(* CoDeSys 2.3.9.50 project: flat.pro *)
(* Libraries: COMlibV2.lb6 25.2.14 08:37:08, TcpIp.lib 9.1.14 13:33:22, TcBase.lib 14.5.09 11:14:08, TcSystem.lib 7.6.16 10:01:22, ModbusRTU.lib 13.5.15 12:38:16, TcIoFunctions.lib 27.1.17 16:22:22, TcUtilities.lib 3.2.16 15:08:58, STANDARD.LIB 5.6.98 11:03:02 *)

(* Task configuration *)
TASK Standard (PRIORITY := 0, INTERVAL := T#50ms);
	MAIN
END_TASK

(* Global variable list: Global_Variables *)
VAR_GLOBAL

	Clear						: ClearComBuffer;
	MB							: ModbusRtuMaster_KL6x22B;
	TxBufferCom1				: ComBuffer;
	RxBufferCom1				: ComBuffer;
	SerialLineControlCom1			: SerialLineControl;
	ReceiveDataCom1			: ReceiveData;
	SendDataCom1				: SendData;

	iobroker	: iobroker_Struct;
	mqtt_set:			ST_MqttSettings;


	HW_trans_power						AT	%QX0.1:BOOL:=FALSE; (*Подача тока на трансформатор и реле ТЭН-а *)
	HW_vent_in_heat						AT	%QX0.2:BOOL:=FALSE; (* Подогрев притока - ТЭН *)

	HW_vent_in_trans_105_130				AT	%QX0.3:BOOL:=FALSE;  (* Напряжение 110 или 130 В *)
	HW_vent_in_trans_160_220				AT	%QX0.4:BOOL:=TRUE;  (* Напряжение 160 или 220 В *)
	HW_vent_in_trans_LO_HI				AT	%QX0.5:BOOL:=FALSE;  (* Напряжение 110/130  или 160/220 В *)
	HW_steam							AT	%QX0.6:BOOL:=FALSE; (* Разрешение включения увлажнителя *)

	HW_vent_out							AT	%QX0.7:BOOL:=FALSE; (* Вытяжной вентилятор*)
	HW_kitchen_vent_out					AT	%QX1.0:BOOL:=FALSE; (*Надплитная вытяжка*)
	HW_vent_in_heat_level				AT	%QX1.1:BOOL:=FALSE; (* Подогрев притока ночной режим   -5 К ТЭН *)
	HW_vent_valve						AT	%QX1.2:BOOL:=FALSE; (*Клапан приточной вентиляции"*)

	HW_valve_water_kitchen				AT	%QX1.3:BOOL; (* Кран ХВС и ГВС на кухне *)
	HW_valve_water_bathroom				AT	%QX1.4:BOOL; (* Кран ХВС и ГВС в санузле *)
	HW_LIGHT_ALL						AT	%QX1.5:BOOL; (*Свет в квартире *)
	HW_LIGHT_hall						AT	%QX1.6:BOOL:=FALSE; (*Ночной/аварийный свет в коридоре *)


	HW_sensor_fld_kitchen				AT %IX0.0:BOOL; (* Датчик протечки на кухне*)
	HW_sensor_fld_tlt						AT %IX0.1:BOOL; (* Датчик протечки в туалете*)
	HW_sensor_fld_post					AT %IX0.2:BOOL; (* Датчик протечки в постирочной*)
	HW_sensor_fld_van					AT %IX0.3:BOOL; (* Датчик протечки в ванной*)
	HW_impulse_kitchen_water_warm		AT %IX0.5:BOOL; (* Счётчик горячей воды на кухне*)
	HW_impulse_kitchen_water_cold		AT %IX0.4:BOOL; (* Счётчик холодной воды на кухне*)
	HW_vent_reay_pressure				AT %IX0.6:BOOL; (*Реле давления*)
	HW_kitchen_button_vent_out			AT %IX0.7:BOOL; (* Кнопка кухонной вытяжки*)

	HW_sensor_vent_valve_opened		AT %IX1.0:BOOL;
	HW_sensor_vent_valve_closed			AT %IX1.1:BOOL;
	HW_impulse_bathroom_water_cold		AT %IX1.2:BOOL; (* Счётчик горячей воды санузла NAMUR*)
	HW_impulse_bathroom_water_warm		AT %IX1.3:BOOL; (* Счётчик холодной воды санузла NAMUR*)
	HW_IN01							AT %IX1.4:BOOL;(*Кнопка вкл и откл света в квартире*)
	HW_IN02							AT %IX1.5:BOOL;(*Кнопка вкл и откл кранов воды на кухне*)
	HW_IN03							AT %IX1.6:BOOL;(*Кнопка вкл и откл кранов воды на кухне*)
	HW_IN04							AT %IX1.7:BOOL;(*Кнопка вкл и откл Вентиляции*)
	HW_IN05							AT %IX2.0:BOOL;(*Кнопка вкл и откл Резерв*)

	HW_gerkon							AT %IX2.1:BOOL;(*Датчик открытия двери - геркон*)
	HW_PIR_door						AT %IX2.2:BOOL;(*Датчик открытия двери - pir *)
	HW_PIR_hall							AT %IX2.3:BOOL;(*Датчик открытия двери - pir *)



	HW_vent_out_level					AT	%QW4:WORD:=7000;(* Напряжение управления вытяжным вентилятором (0-32767) *)

	HW_temp_kitchen_box					AT %IW32:WORD; (*Температура на кухне в коробе  *)
	HW_temp_vent_in						AT %IW34:WORD; (*Температура притока перед фильтром *)
	HW_temp_street						AT %IW36:WORD; (*Температура на улице *)
	HW_temp_bedroom					AT %IW38:WORD; (*Температура в спальне *)


END_VAR

(* Global variable list: Global_Variables_persistent *)
VAR_GLOBAL PERSISTENT

	(*USER VARIABLES NEED TO BE ATTACHED TO %Q TO ENABLE SAVE IT IN NOVRAM, FOR CX ONLY *)

	Target_hum_mem		AT %Q*:		INT;
	Target_CO2_mem		AT %Q*:		INT;
	Vent_mem			AT %Q*:		BOOL;
	Vent_out_mem		AT %Q*:		BOOL;
	Vent_heat_mem		AT %Q*:		INT;
	Steam_mem			AT %Q*:		BOOL;
	Vent_heat_level_mem	AT %Q*:		BOOL;
	Light_mem			AT %Q*:		BOOL; (*Свет в квартире*)

	Kitchen_stat_cold_water_mem		AT %Q*:		DINT;
	Kitchen_stat_warm_water_mem		AT %Q*:		DINT;
	Bathroom_stat_cold_water_mem		AT %Q*:		DINT;
	Bathroom_stat_warm_water_mem	AT %Q*:		DINT;


END_VAR

(* Global variable list: TwinCAT_Configuration *)
(* Generated automatically by TwinCAT - (read only) *)
VAR_CONFIG
	.Target_hum_mem AT %QB36 : INT;
	.Target_CO2_mem AT %QB38 : INT;
	.Vent_mem AT %QX60.0 : BOOL;
	.Vent_out_mem AT %QX60.1 : BOOL;
	.Vent_heat_mem AT %QB40 : INT;
	.Steam_mem AT %QX60.2 : BOOL;
	.Vent_heat_level_mem AT %QX60.3 : BOOL;
	.Light_mem AT %QX60.4 : BOOL;
	.Kitchen_stat_cold_water_mem AT %QB44 : DINT;
	.Kitchen_stat_warm_water_mem AT %QB48 : DINT;
	.Bathroom_stat_cold_water_mem AT %QB52 : DINT;
	.Bathroom_stat_warm_water_mem AT %QB56 : DINT;
END_VAR

(* Global variable list: Variable_Configuration *)
VAR_CONFIG
	MB.InData AT %IB12 : MB_KL6inData22B;
	MB.OutData AT %QB12 : MB_KL6outData22B;
END_VAR

(* Data type *)
TYPE iobroker_Struct  :
STRUCT
	Vent_status				: 	INT;
	Valve_status				: 	INT;
	Kitchen_room_temp 		:	REAL;
	Kitchen_room_hum 		:	REAL;
	Kitchen_room_CO2		:	REAL;

	Child_small_room_temp 	:	REAL;
	Child_small_room_hum 	:	REAL;
	Child_small_room_CO2 	:	REAL;

	Child_big_room_temp	 	:	REAL;
	Child_big_room_hum	 	:	REAL;
	Child_big_room_CO2	 	:	REAL;

	Bed_room_temp	 		:	REAL;
	Bed_room_temp2	 		:	REAL;
	Bed_room_hum	 		:	REAL;
	Bed_room_hum2	 		:	REAL;
	Bed_room_CO2			:	REAL;

	Kitchen_room_tempout		:	REAL;
	Kitchen_room_tempout_2	:	REAL;

	FLD_valve_kitchen 		:	BOOL; (* Положение  крана воды на кухне*)
	FLD_valve_bathroom 		:	BOOL; (*Положение  крана воды в санузле*)
	FLD_PRC				:	BOOL; (*Датчик в постирочной*)
	FLD_TLT				:	BOOL; (*Датчик в туалете*)
	FLD_BATH				:	BOOL;(*Датчик в  ванной*)
	FLD_KUH				:	BOOL;(*Датчик на  кухне*)
	FLD_ALRM_KITCHEN 		:	BOOL; (*ТРЕВОГА ЗАТОПЛЕНИЕ НА КУХНЕ*)
	FLD_ALRM_BATH 		:	BOOL; (*ТРЕВОГА ЗАТОПЛЕНИЕ В САНУЗЛЕ*)


	Kitchen_stat_cold_water	:	DINT;
	Kitchen_stat_warm_water	:	DINT;
	Bathroom_stat_cold_water	:	DINT;
	Bathroom_stat_warm_water	:	DINT;

	Steam_status				:	INT;
	Steam_real				:	INT;

	Vent_input_level			:	INT;  (*  0-220 V  *)
	Vent_output_level			:	INT; (*0-100%*)
	Soft_kitchen_button_vent_out:	BOOL; (*Вирутальная  кнопка кухонной вытяжки*)

	Temp_vent_in			:	REAL;
	Vent_pressure_relay		:	BOOL;

	PT_temp_bedroom		:	REAL;
	Vent_valve_status			:	INT;


	(* SETTINGS *)
	Rezerv					:	BOOL;
	Steam_level				:	INT;
	Security_status			:	INT;
	Target_hum				:	INT;
	Target_CO2				:	INT;
	Vent						:	BOOL;
	Vent_out					:	BOOL;
	Vent_heat				:	INT;
	Steam					:	BOOL;
	Vent_heat_level			:	BOOL;
	Light					:	BOOL; (*Свет в квартире*)
	Light_hall				:	BOOL; (*Свет в коридоре*)
	Gerkon					:	BOOL; (*Датчик открытия входной двери (геркон)*)
	PIR_door				:	BOOL;(*Датчик открытия входной двери PIR-штора*)

	Uv						:	REAL;
	Ia						:	REAL;
	Pw						:	REAL;
	E_T1					:	REAL;
	E_T2					:	REAL;
	E_T4					:	REAL;

END_STRUCT
END_TYPE

(* Data type *)
(* @NESTEDCOMMENTS := 'Yes' *)
(* @PATH := '' *)
(* @OBJECTFLAGS := '0, 8' *)
TYPE ST_MqttReceivedPublishTelegram :
STRUCT
	sTopic		: STRING[255];
	sValue		: STRING[255];
	bHasData	: BOOL;
END_STRUCT
END_TYPE
(* @END_DECLARATION := '0' *)

(* Data type *)
(* @NESTEDCOMMENTS := 'Yes' *)
(* @PATH := '' *)
(* @OBJECTFLAGS := '0, 8' *)
TYPE ST_MqttSettings :
STRUCT
	(* informations *)
(*	sMqttClientId	: STRING[23]:='plc';
	sMqttUserId	: STRING[25]:='mqtt';
	sMqttPassword	: STRING[25]:='mqtt';
	sMqttBrokerIP	: STRING[15]:='192.168.3.200';
	nMqttBrokerPort	: UDINT := 1883;

	(* state *)
	bSocketConnection	: BOOL := FALSE;
	bConnected			: BOOL := FALSE;
	bConnectPackageSent	: BOOL := FALSE;
	bDisconnect			: BOOL := FALSE;
	bError				: BOOL := FALSE;
	bValidConnection	: BOOL := FALSE;
	bActive				: BOOL := FALSE;
	wPackageIdentifier	: WORD := 1;
	hSocket				: T_HSOCKET;
	tonSendPingReq		: TON;

	(* send *)
	stMqttSendTelegram			: ST_MqttTelegram;
	stMqttLastSendTelegram		: ST_MqttTelegram;

	(* receive *)
	stMqttReceivedTelegram			: ST_MqttTelegram;
	stMqttLastReceivedTelegram		: ST_MqttTelegram;
	stMqttReceivedPublishTelegram	: ST_MqttReceivedPublishTelegram;

	(* settings internal *)
	iTelegramSize	: INT := 544;
	usKeepAliveTime	: USINT := 60; (* seconds *)

*)



	(* informations *)
	sMqttClientId	: STRING[23];
	sMqttUserId	: STRING[25];
	sMqttPassword	: STRING[25];
	sMqttBrokerIP	: STRING[15];
	nMqttBrokerPort	: UDINT := 1883;

	(* state *)
	bSocketConnection	: BOOL := FALSE;
	bConnected			: BOOL := FALSE;
	bConnectPackageSent	: BOOL := FALSE;
	bDisconnect			: BOOL := FALSE;
	bError				: BOOL := FALSE;
	bValidConnection	: BOOL := FALSE;
	bActive				: BOOL := FALSE;
	wPackageIdentifier	: WORD := 1;
	hSocket				: T_HSOCKET;
	tonSendPingReq		: TON;

	(* send *)
	stMqttSendTelegram			: ST_MqttTelegram;
	stMqttLastSendTelegram		: ST_MqttTelegram;

	(* receive *)
	stMqttReceivedTelegram			: ST_MqttTelegram;
	stMqttLastReceivedTelegram		: ST_MqttTelegram;
	stMqttReceivedPublishTelegram	: ST_MqttReceivedPublishTelegram;

	(* settings internal *)
	iTelegramSize	: INT := 544;
	usKeepAliveTime	: USINT := 60; (* seconds *)










END_STRUCT
END_TYPE
(* @END_DECLARATION := '0' *)

(* Data type *)
(* @NESTEDCOMMENTS := 'Yes' *)
(* @PATH := '' *)
(* @OBJECTFLAGS := '0, 8' *)
TYPE ST_MqttTelegram :
STRUCT
	arMqttData 	: ARRAY[0..544] OF BYTE;
	nDataLength	: UDINT := 0;
END_STRUCT
END_TYPE
(* @END_DECLARATION := '0' *

(* POU MAIN, ST *)
PROGRAM MAIN
VAR
	INITVAR					: BOOL:=FALSE;
	SW_LIGHT				: SM_BUTT;		(* вкл/откл  света в квартире *)
	SW_VENT				: SM_BUTT;		(* вкл/откл вентиляции *)
	SW_REZERV			: SM_BUTT;





END_VAR
IF (INITVAR=FALSE) THEN

(* RESTORE VARS FROM MEMORY AFTER REBOOT/RESET/LOST POWER *)

	iobroker.Target_hum		:=	Target_hum_mem;
	iobroker.Target_CO2		:=	Target_CO2_mem;
	iobroker.Vent				:=	Vent_mem;
	iobroker.Vent_out			:=	Vent_out_mem;
	iobroker.Vent_heat		:=	Vent_heat_mem;
	iobroker.Steam			:=	Steam_mem;
	iobroker.Vent_heat_level	:=	Vent_heat_level_mem;
	iobroker.Light				:=	Light_mem;

	iobroker.Kitchen_stat_cold_water		:=	Kitchen_stat_cold_water_mem;
	iobroker.Kitchen_stat_warm_water		:=	Kitchen_stat_warm_water_mem;
	iobroker.Bathroom_stat_cold_water		:=	Bathroom_stat_cold_water_mem;
	iobroker.Bathroom_stat_warm_water		:=	Bathroom_stat_warm_water_mem;

	INITVAR:=TRUE;
ELSE

	(* SAVE VARS to PERSISTENT *)

	Target_hum_mem		:=	iobroker.Target_hum;
	Target_CO2_mem		:=	iobroker.Target_CO2;
	Vent_mem			:=	iobroker.Vent;
	Vent_out_mem		:=	iobroker.Vent_out;
	Vent_heat_mem		:=	iobroker.Vent_heat;
	Steam_mem			:=	iobroker.Steam;
	Vent_heat_level_mem	:=	iobroker.Vent_heat_level;
	Light_mem			:=	iobroker.Light;

	Mqtt;					(*Отправка данных mqtt *)
	Sensors;					(* Аналоговые датчики на модуле KL *)
	RS485read;				(* Работа с устройствами на шине RS485 *)
	VentControl;				(* Глобальный контроль вентустановки*)
	VentPower;				(* Авторегулировка мощности вентустановки по датчикам CO2*)
	Counters;				(* Счётчики воды *)
	Fluid_bath;				(* Защита от протечки в санузлах. Оработка нажатия физической и виртульной кнопки №2 *)
	Fluid_kitchen;				(* Защита от протечки в кухне. Оработка нажатия физической и виртульной кнопки №3 *)
	Light_hall;				(* Свет в коридоре *)



(* Оработка нажатия физических и виртульных кнопок №1, №4, №5 *)

	SW_LIGHT 		(IN:=HW_IN01, IN1:= iobroker.Light, 	Q=>NOT iobroker.Light);	(* Конпка №1 *)
	SW_VENT 		(IN:=HW_IN04, IN1:=iobroker.Vent, 	Q=>iobroker.Vent);		(* Конпка №4 *)
	SW_REZERV 	(IN:=HW_IN05, IN1:=iobroker.Rezerv, 	Q=>iobroker.Rezerv);	(* Конпка №5 *)


(* Прямая связь между экспортирумымми переменными и  переменными, жестко привязаными  к физ. портам. Частота обновления= циклу ПЛК  : *)

	HW_LIGHT_ALL	:=NOT iobroker.Light;					(* СВЕТ в квартире*)
	HW_LIGHT_HALL	:=iobroker.Light_hall;					(* СВЕТ в квартире*)
	iobroker.Gerkon	:=HW_gerkon;						(* Геркон на двери*)
	iobroker.PIR_door:=HW_pir_door;						(* Датчик движения на двери *)
	iobroker.Vent_pressure_relay:=HW_vent_reay_pressure; 	(* Relay pressure *)

END_IF
END_PROGRAM

(* POU SM_BUTT, ST *)
FUNCTION_BLOCK SM_BUTT            (* ФУНКЦИОНАЛЬНЫЙ БЛОК ДЛЯ ПРОСТОЙ КНОПКИ *)
    VAR_INPUT
       	IN: BOOL;          	(*ВХОД ЗА КОТОРЫМ МЫ СЛЕДИМ *)
	IN1:BOOL;				(*ВЫХОД ЗА КОТОРЫМ ТОЖЕ СЛЕДИМ*)
    END_VAR

    VAR_OUTPUT
	Q : BOOL;        			(*СОСТОЯНИЕ ВЫХОДА*)
    END_VAR
    VAR
  MEM : BOOL;    			(* ВНУТРЕННЯЯ ПЕРЕМЕННАЯ ДЛЯ ХРАНЕНИЯ СОСТОЯНИЯ КНОПКИ *)
    END_VAR
Q:=IN1;

IF IN AND NOT MEM THEN 	(* ПОЙМАЛИ ПЕРЕДНИЙ ФРОНТ - НАЖАЛИ НА КНОПКУ *)
	Q := NOT IN1;    			(* МЕНЯЕМ СОСТОЯНИЕ ВЫХОДА НА ПРОТИВОПОЛОЖНОЕ *)
END_IF

MEM := IN;                       		(* ЗАПОМИНАЕМ ТЕКУЩЕЕ ЗНАЧЕНИЕ КНОПКИ *)
END_FUNCTION_BLOCK

(* POU Mqtt, ST *)
PROGRAM Mqtt
VAR
	FB_Mqtt_Controller 		: FB_Mqtt_Controller_V10;
	stMqttSettings				: ST_MqttSettings;
	bMqttControllerBusy		: BOOL;
	FB_Mqtt_Publish1 			: FB_Mqtt_Publish_V10;
	FB_Mqtt_Publish2			: FB_Mqtt_Publish_V10;
	FB_Mqtt_Publish3			: FB_Mqtt_Publish_V10;
	FB_Mqtt_Publish4			: FB_Mqtt_Publish_V10;
	bPublishBusy1			: BOOL;
	bPublishBusy2			: BOOL;
	bPublishBusy3			: BOOL;
	bPublishBusy4			: BOOL;
END_VAR
(*        SEND DATA VIA MQTT  *)

FB_Mqtt_Controller (
		bActive			:= TRUE,
		sMqttClientId		:= 'plc',
		sMqttUserId		:= 'mqtt',
		sMqttPassword	:= 'mqtt',
		sMqttBrokerIp		:= '192.168.3.200',
		nMqttBrokerPort	:= 1883,
		stMqttSettings		:= stMqttSettings,
		bBusy			=> bMqttControllerBusy
	);
	IF bMqttControllerBusy THEN
		RETURN;
	END_IF

		FB_Mqtt_Publish1(sTopic:='BECKHOFF_CX9010/CO2/Kitchen',sValue:=REAL_TO_STRING(iobroker.Kitchen_room_CO2),bRetain:=TRUE, stMqttSettings:=stMqttSettings,bBusy => bPublishBusy1 );
		FB_Mqtt_Publish2(sTopic:='BECKHOFF_CX9010/CO2/Bed_room',sValue:=REAL_TO_STRING(iobroker.Bed_room_CO2),bRetain:=TRUE, stMqttSettings:=stMqttSettings,bBusy => bPublishBusy2 );
		FB_Mqtt_Publish3(sTopic:='BECKHOFF_CX9010/CO2/Child_big_room',sValue:=REAL_TO_STRING(iobroker.Child_big_room_CO2),bRetain:=TRUE, stMqttSettings:=stMqttSettings,bBusy => bPublishBusy3 );
		FB_Mqtt_Publish4(sTopic:='BECKHOFF_CX9010/CO2/Child_small_room',sValue:=REAL_TO_STRING(iobroker.Child_small_room_CO2),bRetain:=TRUE, stMqttSettings:=stMqttSettings,bBusy => bPublishBusy4);
END_PROGRAM

(* POU FB_Mqtt_Controller_V10, ST *)
(* @NESTEDCOMMENTS := 'Yes' *)
(* @PATH := '\/_Generic\/Mqtt' *)
(* @OBJECTFLAGS := '0, 8' *)
(* @SYMFILEFLAGS := '2048' *)
FUNCTION_BLOCK FB_Mqtt_Controller_V10
VAR_INPUT
(*	bActive			: BOOL := FALSE;
	sMqttClientId	: STRING[23]:='plc';
	sMqttUserId	: STRING[25] := 'mqtt';
	sMqttPassword	: STRING[25] := 'mqtt';
	sMqttBrokerIP	: STRING[15]:='192.168.3.200';
	nMqttBrokerPort	: UDINT := 1883;
*)
	bActive			: BOOL := FALSE;
	sMqttClientId	: STRING[23];
	sMqttUserId	: STRING[25] := '';
	sMqttPassword	: STRING[25] := '';
	sMqttBrokerIP	: STRING[15];
	nMqttBrokerPort	: UDINT := 1883;
END_VAR
VAR_OUTPUT
	bBusy	: BOOL := FALSE;
END_VAR
VAR_IN_OUT
	stMqttSettings	: ST_MqttSettings;
END_VAR
VAR
	iState			: INT := 0;
	fbSocketConnect	: FB_SocketConnect;
	fbSocketClose	: FB_SocketClose;

	fbMqttTelegramConnect	: FB_MqttTelegram_Connect_V10;
	fbMqttTelegramPingReq	: FB_MqttTelegram_PingReq_V10;
	fbMqttSend				: FB_Mqtt_Send_V10;
	fbMqttReceive			: FB_Mqtt_Receive_V10;
END_VAR
VAR CONSTANT
	C_STARTUP					: INT := 0;
	C_CONNECT					: INT := 100;
	C_CONNECT_WAIT				: INT := 110;
	C_CLOSE						: INT := 200;
	C_CLOSE_WAIT				: INT := 210;
	C_IDLE						: INT := 500;
END_VAR
(* @END_DECLARATION := '0' *)
(*
 * Connects to mqtt broker
 * Sends connect message
 * Sends ping(back)
 * Sends disconnect
 *)
CASE iState OF
	C_STARTUP:
		stMqttSettings.bConnected			:= FALSE;
		stMqttSettings.bConnectPackageSent	:= FALSE;
		stMqttSettings.bDisconnect			:= FALSE;
		stMqttSettings.bSocketConnection	:= FALSE;
		stMqttSettings.bError				:= FALSE;
		stMqttSettings.bValidConnection		:= FALSE;
		stMqttSettings.wPackageIdentifier	:= 1;
		stMqttSettings.bActive				:= bActive;
		stMqttSettings.hSocket				:= fbSocketConnect.hSocket;
		stMqttSettings.nMqttBrokerPort		:= nMqttBrokerPort;
		stMqttSettings.sMqttBrokerIP		:= sMqttBrokerIP;
		stMqttSettings.sMqttClientId		:= sMqttClientId;
		stMqttSettings.sMqttUserId		:= sMqttUserId;
		stMqttSettings.sMqttPassword		:= sMqttPassword;

		stMqttSettings.stMqttReceivedTelegram.nDataLength := 0;

		bBusy := FALSE;

		CallMqttBlocks();

		IF bActive THEN
			iState := C_CONNECT;
		END_IF;

	(* Start connection *)
	C_CONNECT:
		bBusy := TRUE;

		fbSocketConnect(
			bExecute	:= FALSE
		);

		fbSocketConnect(
			sSrvNetId	:= '',
			sRemoteHost	:= sMqttBrokerIP,
			nRemotePort	:= nMqttBrokerPort,
			bExecute	:= TRUE,
			tTimeout	:= USINT_TO_TIME(stMqttSettings.usKeepAliveTime) + t#10s
		);

		iState := C_CONNECT_WAIT;

	(* Wait till connected *)
	C_CONNECT_WAIT:
		fbSocketConnect(
			bExecute := FALSE
		);

		IF
			NOT fbSocketConnect.bBusy
			AND NOT fbSocketConnect.bError
		THEN
			iState 								:= C_IDLE;
			stMqttSettings.hSocket				:= fbSocketConnect.hSocket;
			stMqttSettings.bSocketConnection	:= TRUE;
		END_IF;

		IF fbSocketConnect.bError THEN
			iState := C_STARTUP;
		END_IF;

		IF NOT stMqttSettings.bActive THEN
			iState := C_STARTUP;
		END_IF;

	(* Close connection *)
	C_CLOSE:
		bBusy := TRUE;

		fbSocketClose(
			bExecute	:= TRUE,
			hSocket		:= stMqttSettings.hSocket
		);

		iState := C_CLOSE_WAIT;

	(* Wait close connection *)
	C_CLOSE_WAIT:
		fbSocketClose(
			bExecute := FALSE
		);

		IF
			NOT fbSocketClose.bBusy
			AND NOT fbSocketClose.bError
		THEN
			iState := C_STARTUP;
		END_IF;

		IF fbSocketClose.bError THEN
			iState := C_STARTUP;
		END_IF;

		IF NOT stMqttSettings.bActive THEN
			iState := C_STARTUP;
		END_IF;

	(* Idle *)
	C_IDLE:
		bBusy 					:= FALSE;
		stMqttSettings.bActive	:= bActive;

		stMqttSettings.bValidConnection :=
			NOT stMqttSettings.bError
			AND NOT stMqttSettings.bDisconnect
			AND stMqttSettings.bConnected
			AND stMqttSettings.bSocketConnection
			AND stMqttSettings.bActive;

		CallMqttBlocks();

		IF
			stMqttSettings.bDisconnect
			OR stMqttSettings.bError
			OR NOT stMqttSettings.bActive
		THEN
			IF
				stMqttSettings.bConnected
				OR stMqttSettings.bSocketConnection
			THEN
				(* TODO : send disconnect *)
				iState := C_CLOSE;
			ELSE
				iState := C_CLOSE;
			END_IF;
		END_IF;

	ELSE
		iState := C_STARTUP;
END_CASE;
(*	END_FUNCTION_BLOCK	*)
END_FUNCTION_BLOCK
ACTION CallMqttBlocks:
(*ACTION	CallMqttBlocks: *)
fbMqttReceive(
	stMqttSettings := stMqttSettings
);

fbMqttTelegramConnect(
	stMqttSettings := stMqttSettings
);

fbMqttTelegramPingReq(
	stMqttSettings := stMqttSettings
);

fbMqttSend(
	stMqttSettings := stMqttSettings
);

(* END_ACTION *)
END_ACTION

(* POU Intern/FB_MqttTelegram_Connect_V10, ST *)
(* @NESTEDCOMMENTS := 'Yes' *)
(* @PATH := '\/_Generic\/Mqtt\/Intern' *)
(* @OBJECTFLAGS := '0, 8' *)
(* @SYMFILEFLAGS := '2048' *)
FUNCTION_BLOCK FB_MqttTelegram_Connect_V10
VAR_IN_OUT
	stMqttSettings	: ST_MqttSettings;
END_VAR
VAR
	iState 				: INT := 0;
	idLength			: INT;
	iuLength			: INT;
	ipLength			: INT;
	ipos				: INT;
	stMqttTelegram		: ST_MqttTelegram;
	fbMqttEncodeLength	: FB_Mqtt_EncodeLength_V10;
	bLength1			: BYTE;
	bLength2			: BYTE;
	bLength3			: BYTE;
	bLength4			: BYTE;
	bLengthAmount		: BYTE;
END_VAR
VAR CONSTANT
	C_STARTUP		: INT := 0;
	C_BUILD_CONNECT	: INT := 100;
	C_SEND_WAIT		: INT := 110;
	C_IDLE			: INT := 500;
END_VAR
(* @END_DECLARATION := '0' *)
CASE iState OF
	C_STARTUP:
		IF
			NOT stMqttSettings.bDisconnect
			AND NOT stMqttSettings.bError
			AND stMqttSettings.bSocketConnection
			AND stMqttSettings.bActive
		THEN
			iState := C_IDLE;
		END_IF;

	(* build connect telegram *)
	C_BUILD_CONNECT:
		FC_Mqtt_ClearTelegram_V10(
			stMqttTelegram	:= stMqttTelegram,
			stMqttSettings	:= stMqttSettings
		);

		(* get client id length *)
		idLength := LEN(stMqttSettings.sMqttClientId);
		IF idLength < 1 THEN
			stMqttSettings.sMqttClientId := 'x';
			idLength := 1;
		END_IF;

		IF idLength > 23 THEN
			idLength := 23;
		END_IF;

		IF
			LEN(stMqttSettings.sMqttUserId) > 0
			AND LEN(stMqttSettings.sMqttPassword) > 0
		THEN
			iuLength := LEN(stMqttSettings.sMqttUserId)+2; (* 2 byte data length*)
			ipLength := LEN(stMqttSettings.sMqttPassword)+2; (* 2 byte data length*)
		ELSE
			iuLength := 0;
			ipLength := 0;
		END_IF

		(* Calculate length *)
		(* 10 byte header, 2 byte data length, data length, [user length + 2], [password length + 2]*)
		fbMqttEncodeLength(
			dwLength := 10 + 2 + INT_TO_BYTE(idLength) + INT_TO_BYTE(iuLength) + INT_TO_BYTE(ipLength),
			bLength1 => bLength1,
			bLength2 => bLength2,
			bLength3 => bLength3,
			bLength4 => bLength4,
			bAmount	 => bLengthAmount
		);

		(* MQTT Control Packet type *)
		stMqttTelegram.arMqttData[0] := 16;
		(* Remaining Length *)
		CASE bLengthAmount OF
			1:
				stMqttTelegram.arMqttData[1] := bLength1;

			2:
				stMqttTelegram.arMqttData[1] := bLength1;
				stMqttTelegram.arMqttData[2] := bLength2;

			3:
				stMqttTelegram.arMqttData[1] := bLength1;
				stMqttTelegram.arMqttData[2] := bLength2;
				stMqttTelegram.arMqttData[3] := bLength3;

			4:
				stMqttTelegram.arMqttData[1] := bLength1;
				stMqttTelegram.arMqttData[2] := bLength2;
				stMqttTelegram.arMqttData[3] := bLength3;
				stMqttTelegram.arMqttData[4] := bLength4;
		END_CASE;
		(* init position*)
		ipos := bLengthAmount;

		(* Length MSB *)
		stMqttTelegram.arMqttData[ipos+1] := 0;
		(* Length LSB *)
		stMqttTelegram.arMqttData[ipos+2] := 4;
		(* M *)
		stMqttTelegram.arMqttData[ipos+3] := 77;
		(* Q *)
		stMqttTelegram.arMqttData[ipos+4] := 81;
		(* T *)
		stMqttTelegram.arMqttData[ipos+5] := 84;
		(* T *)
		stMqttTelegram.arMqttData[ipos+6] := 84;
		(* Protocol Level *)
		stMqttTelegram.arMqttData[ipos+7] := 4;
		(* Connect Flags *)
		stMqttTelegram.arMqttData[ipos+8].1 := TRUE;
		stMqttTelegram.arMqttData[ipos+8].6 := (ipLength>2); (* more then 2 byte data length*)
		stMqttTelegram.arMqttData[ipos+8].7 := (iuLength>2); (* more then 2 byte data length*)
		(* Keep Alive MSB *)
		stMqttTelegram.arMqttData[ipos+9] := 0;
		(* Keep Alive LSB *)
		stMqttTelegram.arMqttData[ipos+10] := stMqttSettings.usKeepAliveTime;
		(* Data length MSB *)
		stMqttTelegram.arMqttData[ipos+11] := 0;
		(* Data length LSB *)
		stMqttTelegram.arMqttData[ipos+12] := INT_TO_BYTE(idLength);

		(* Client ID *)
		MEMCPY(
			destAddr	:= ADR(stMqttTelegram.arMqttData[ipos+13]),
		    srcAddr		:= ADR(stMqttSettings.sMqttClientId),
			n  			:= idLength
		);

		ipos := ipos+13+idLength;
		IF (iuLength > 2) THEN (* more then 2 byte data length*)
			(* Data length MSB *)
			stMqttTelegram.arMqttData[ipos] := 0;
			(* Data length LSB *)
			stMqttTelegram.arMqttData[ipos+1] := INT_TO_BYTE(iuLength-2);

			(* User ID *)
			MEMCPY(
				destAddr	:= ADR(stMqttTelegram.arMqttData[ipos+2]),
			    srcAddr		:= ADR(stMqttSettings.sMqttUserId),
				n  			:= iuLength-2
			);
			ipos := ipos+iuLength;
		END_IF

		IF (iuLength > 2) THEN (* more then 2 byte data length*)
			(* Data length MSB *)
			stMqttTelegram.arMqttData[ipos] := 0;
			(* Data length LSB *)
			stMqttTelegram.arMqttData[ipos+1] := INT_TO_BYTE(ipLength-2);

			(* Password *)
			MEMCPY(
				destAddr	:= ADR(stMqttTelegram.arMqttData[ipos+2]),
			    srcAddr		:= ADR(stMqttSettings.sMqttPassword),
				n  			:= ipLength-2
			);
			ipos := ipos+ipLength;
		END_IF

		stMqttTelegram.nDataLength 	:= ipos; (* 1 byte header, 1 byte remaining length *)
		iState 						:= C_SEND_WAIT;

	(* send telegram *)
	C_SEND_WAIT:
		IF stMqttSettings.stMqttSendTelegram.nDataLength = 0 THEN
			FC_Mqtt_CopyTelegram_V10(
				stMqttSrcTelegram	:= stMqttTelegram,
				stMqttDestTelegram	:= stMqttSettings.stMqttSendTelegram,
				stMqttSettings		:= stMqttSettings
			);

			stMqttSettings.bConnectPackageSent	:= TRUE;
			iState								:= C_IDLE;
		END_IF;

		IF
			NOT stMqttSettings.bActive
			OR NOT stMqttSettings.bSocketConnection
		THEN
			iState := C_STARTUP;
		END_IF;

	(* idle *)
	C_IDLE:
		IF
			NOT stMqttSettings.bDisconnect
			AND NOT stMqttSettings.bError
			AND NOT stMqttSettings.bConnected
			AND stMqttSettings.bSocketConnection
			AND NOT stMqttSettings.bConnectPackageSent
			AND stMqttSettings.bActive
		THEN
			iState := C_BUILD_CONNECT;
		END_IF;

		(* check received telegram *)
		IF
			stMqttSettings.bConnectPackageSent
			AND stMqttSettings.stMqttReceivedTelegram.nDataLength = 4
			AND stMqttSettings.stMqttReceivedTelegram.arMqttData[0] = 32
			AND stMqttSettings.stMqttReceivedTelegram.arMqttData[1] = 2
			AND (
				(* Session pressent or not, we ignore *)
				stMqttSettings.stMqttReceivedTelegram.arMqttData[2] = 1
				OR
				stMqttSettings.stMqttReceivedTelegram.arMqttData[2] = 0
			)
			AND stMqttSettings.stMqttReceivedTelegram.arMqttData[3] = 0
		THEN
			stMqttSettings.bConnected := TRUE;
			FC_Mqtt_ClearTelegram_V10(
				stMqttTelegram	:= stMqttSettings.stMqttReceivedTelegram,
				stMqttSettings	:= stMqttSettings
			);
		END_IF;

		(* error on connect *)
		IF
			stMqttSettings.bConnectPackageSent
			AND stMqttSettings.stMqttReceivedTelegram.nDataLength = 4
			AND stMqttSettings.stMqttReceivedTelegram.arMqttData[0] = 32
			AND stMqttSettings.stMqttReceivedTelegram.arMqttData[1] = 2
			AND stMqttSettings.stMqttReceivedTelegram.arMqttData[3] <> 0
		THEN
			stMqttSettings.bError := TRUE;
		END_IF;

		IF
			stMqttSettings.bDisconnect
			OR stMqttSettings.bError
			OR NOT stMqttSettings.bSocketConnection
			OR NOT stMqttSettings.bActive
		THEN
			iState := C_STARTUP;
		END_IF;

	ELSE
		iState := C_STARTUP;
END_CASE;


(*	END_FUNCTION_BLOCK	*)
END_FUNCTION_BLOCK

(* POU Intern/FB_Mqtt_EncodeLength_V10, ST *)
(* @NESTEDCOMMENTS := 'Yes' *)
(* @PATH := '\/_Generic\/Mqtt\/Intern' *)
(* @OBJECTFLAGS := '0, 8' *)
(* @SYMFILEFLAGS := '2048' *)
FUNCTION_BLOCK FB_Mqtt_EncodeLength_V10
VAR_INPUT
	dwLength	: DWORD;
END_VAR
VAR_OUTPUT
	bLength1	: BYTE := 0;
	bLength2	: BYTE := 0;
	bLength3	: BYTE := 0;
	bLength4	: BYTE := 0;
	bAmount		: BYTE := 0;
END_VAR
VAR
	dwWorkLength	: DWORD;
	dwCopyLength	: DWORD;
END_VAR
(* @END_DECLARATION := '0' *)
bAmount 		:= 1;
dwCopyLength	:= dwLength;

WHILE dwCopyLength > 0 DO
	dwWorkLength := dwCopyLength MOD 128;
	dwCopyLength := dwCopyLength / 128;

	IF dwCopyLength > 0 THEN
		dwWorkLength := dwWorkLength OR 128;
	END_IF;

	CASE bAmount OF
		1:
			bLength1 := DWORD_TO_BYTE(dwWorkLength);

		2:
			bLength2 := DWORD_TO_BYTE(dwWorkLength);

		3:
			bLength3 := DWORD_TO_BYTE(dwWorkLength);

		4:
			bLength4 := DWORD_TO_BYTE(dwWorkLength);

		ELSE
			;
	END_CASE;

	IF dwCopyLength > 0 THEN
		bAmount := bAmount + 1;
	END_IF;

	IF bAmount > 4 THEN
		(* hmm *)
		RETURN;
	END_IF;
END_WHILE;
(*
do
	encodedByte = X MOD 128
	X = X DIV 128

	// if there are more data to encode, set the top bit of this byte
	if ( X > 0 )
		encodedByte = encodedByte OR 128
	endif

	'output' encodedByte
while ( X > 0 )
*)

(*	END_FUNCTION_BLOCK	*)
END_FUNCTION_BLOCK

(* POU Intern/FC_Mqtt_ClearTelegram_V10, ST *)
(* @NESTEDCOMMENTS := 'Yes' *)
(* @PATH := '\/_Generic\/Mqtt\/Intern' *)
(* @OBJECTFLAGS := '0, 8' *)
(* @SYMFILEFLAGS := '2048' *)
FUNCTION FC_Mqtt_ClearTelegram_V10 : BOOL
VAR_IN_OUT
	stMqttTelegram	: ST_MqttTelegram;
	stMqttSettings	: ST_MqttSettings;
END_VAR
VAR
END_VAR
(* @END_DECLARATION := '0' *)
MEMSET(
	destAddr	:= ADR(stMqttTelegram.arMqttData),
	fillByte  	:= 0,
	n			:= stMqttSettings.iTelegramSize
);

stMqttTelegram.nDataLength := 0;

(*	END_FUNCTION	*)
END_FUNCTION

(* POU Intern/FC_Mqtt_CopyTelegram_V10, ST *)
(* @NESTEDCOMMENTS := 'Yes' *)
(* @PATH := '\/_Generic\/Mqtt\/Intern' *)
(* @OBJECTFLAGS := '0, 8' *)
(* @SYMFILEFLAGS := '2048' *)
FUNCTION FC_Mqtt_CopyTelegram_V10 : BOOL
VAR_IN_OUT
	stMqttSrcTelegram	: ST_MqttTelegram;
	stMqttDestTelegram	: ST_MqttTelegram;
	stMqttSettings		: ST_MqttSettings;
END_VAR
VAR
END_VAR
(* @END_DECLARATION := '0' *)
MEMCPY(
	destAddr	:= ADR(stMqttDestTelegram.arMqttData),
    srcAddr		:= ADR(stMqttSrcTelegram.arMqttData),
	n  			:= stMqttSettings.iTelegramSize
);

stMqttDestTelegram.nDataLength := stMqttSrcTelegram.nDataLength;

(*	END_FUNCTION	*)
END_FUNCTION

(* POU Intern/FB_MqttTelegram_PingReq_V10, ST *)
(* @NESTEDCOMMENTS := 'Yes' *)
(* @PATH := '\/_Generic\/Mqtt\/Intern' *)
(* @OBJECTFLAGS := '0, 8' *)
(* @SYMFILEFLAGS := '2048' *)
FUNCTION_BLOCK FB_MqttTelegram_PingReq_V10
VAR_IN_OUT
	stMqttSettings	: ST_MqttSettings;
END_VAR
VAR
	iState 				: INT := 0;
	bMustSend			: BOOL := FALSE;
	bPingReqSent		: BOOL := FALSE;
	stMqttTelegram		: ST_MqttTelegram;
END_VAR
VAR CONSTANT
	C_STARTUP		: INT := 0;
	C_BUILD_PING	: INT := 100;
	C_SEND_WAIT		: INT := 110;
	C_IDLE			: INT := 500;
END_VAR
(* @END_DECLARATION := '0' *)
CASE iState OF
	C_STARTUP:
		bPingReqSent := FALSE;

		IF stMqttSettings.bValidConnection THEN
			iState := C_IDLE;
		END_IF;

	(* build pingreq telegram *)
	C_BUILD_PING:
		FC_Mqtt_ClearTelegram_V10(
			stMqttTelegram	:= stMqttTelegram,
			stMqttSettings	:= stMqttSettings
		);

		(* MQTT Control Packet type *)
		stMqttTelegram.arMqttData[0] := 192;
		(* Remaining Length *)
		stMqttTelegram.arMqttData[1] := 0;

		stMqttTelegram.nDataLength := 2;

		iState := C_SEND_WAIT;

	(* send telegram *)
	C_SEND_WAIT:
		IF stMqttSettings.stMqttSendTelegram.nDataLength = 0 THEN
			FC_Mqtt_CopyTelegram_V10(
				stMqttSrcTelegram	:= stMqttTelegram,
				stMqttDestTelegram	:= stMqttSettings.stMqttSendTelegram,
				stMqttSettings		:= stMqttSettings
			);

			bPingReqSent	:= TRUE;
			iState			:= C_IDLE;
		END_IF;

		IF NOT stMqttSettings.bValidConnection THEN
			iState := C_STARTUP;
		END_IF;

	(* idle *)
	C_IDLE:
		bMustSend := FALSE;

		IF stMqttSettings.usKeepAliveTime > 0 THEN
			bMustSend := stMqttSettings.tonSendPingReq.Q;
		END_IF;

		IF
			stMqttSettings.bValidConnection
			AND bMustSend
			AND NOT bPingReqSent
		THEN
			iState := C_BUILD_PING;
		END_IF;

		(* Check received telegram *)
		IF
			bPingReqSent
			AND stMqttSettings.stMqttReceivedTelegram.nDataLength = 2
			AND stMqttSettings.stMqttReceivedTelegram.arMqttData[0] = 208
			AND stMqttSettings.stMqttReceivedTelegram.arMqttData[1] = 0
		THEN
			FC_Mqtt_ClearTelegram_V10(
				stMqttTelegram	:= stMqttSettings.stMqttReceivedTelegram,
				stMqttSettings	:= stMqttSettings
			);
			bPingReqSent := FALSE;
		END_IF;

		IF NOT stMqttSettings.bValidConnection THEN
			iState := C_STARTUP;
		END_IF;

	ELSE
		iState := C_STARTUP;
END_CASE;

(*	END_FUNCTION_BLOCK	*)
END_FUNCTION_BLOCK

(* POU Intern/FB_Mqtt_Send_V10, ST *)
(* @NESTEDCOMMENTS := 'Yes' *)
(* @PATH := '\/_Generic\/Mqtt\/Intern' *)
(* @OBJECTFLAGS := '0, 8' *)
(* @SYMFILEFLAGS := '2048' *)
FUNCTION_BLOCK FB_Mqtt_Send_V10
VAR_OUTPUT
	bBusy	: BOOL := FALSE;
END_VAR
VAR_IN_OUT
	stMqttSettings	: ST_MqttSettings;
END_VAR
VAR
	fbSocketSend 	: FB_SocketSend;
	tPingReq		: TIME;
	iState 			: INT := 0;
	stSendTelegram	: ST_MqttTelegram;
END_VAR
VAR CONSTANT
	C_STARTUP		: INT := 0;
	C_SEND			: INT := 100;
	C_SEND_WAIT		: INT := 110;
	C_IDLE			: INT := 500;
END_VAR
(* @END_DECLARATION := '0' *)
CASE iState OF
	C_STARTUP:
		bBusy := FALSE;

		stMqttSettings.tonSendPingReq(
			in := FALSE
		);

		IF
			NOT stMqttSettings.bDisconnect
			AND NOT stMqttSettings.bError
			AND stMqttSettings.bSocketConnection
		THEN
			iState := C_IDLE;
		END_IF;

	(* send mqtt telegram *)
	C_SEND:
		bBusy := TRUE;

		(* copy send telegram *)
		FC_Mqtt_CopyTelegram_V10(
			stMqttSrcTelegram	:= stMqttSettings.stMqttSendTelegram,
			stMqttDestTelegram	:= stSendTelegram,
			stMqttSettings		:= stMqttSettings
		);

		(* start send *)
		fbSocketSend(
			bExecute := FALSE
		);

		fbSocketSend(
			sSrvNetId	:= '',
			hSocket		:= stMqttSettings.hSocket,
			cbLen		:= stSendTelegram.nDataLength,
			pSrc		:= ADR(stSendTelegram.arMqttData),
			bExecute 	:= TRUE
		);

		iState := C_SEND_WAIT;

	(* wait send done *)
	C_SEND_WAIT:
		fbSocketSend(
			bExecute := FALSE
		);

		IF
			NOT fbSocketSend.bBusy
			AND NOT fbSocketSend.bError
		THEN
			(* copy last telegram *)
			FC_Mqtt_CopyTelegram_V10(
				stMqttSrcTelegram	:= stMqttSettings.stMqttSendTelegram,
				stMqttDestTelegram	:= stMqttSettings.stMqttLastSendTelegram,
				stMqttSettings		:= stMqttSettings
			);

			(* clear send buffer *)
			FC_Mqtt_ClearTelegram_V10(
				stMqttTelegram 	:= stMqttSettings.stMqttSendTelegram,
				stMqttSettings	:= stMqttSettings
			);

			iState	:= C_IDLE;
			bBusy	:= FALSE;
		END_IF;

		IF stMqttSettings.usKeepAliveTime > 0 THEN
			tPingReq := DWORD_TO_TIME(USINT_TO_DWORD(stMqttSettings.usKeepAliveTime) * 1000 - 5000);

			stMqttSettings.tonSendPingReq(
				in := FALSE
			);

			stMqttSettings.tonSendPingReq(
				in := TRUE,
				pt := tPingReq
			);
		END_IF;

		IF fbSocketSend.bError THEN
			iState 					:= C_STARTUP;
			stMqttSettings.bError	:= TRUE;
		END_IF;

		IF
			NOT stMqttSettings.bActive
			OR NOT stMqttSettings.bSocketConnection
		THEN
			iState := C_STARTUP;
		END_IF;

	(* idle *)
	C_IDLE:
		IF stMqttSettings.usKeepAliveTime > 0 THEN
			stMqttSettings.tonSendPingReq(
				in := stMqttSettings.bConnected
			);
		ELSE
			stMqttSettings.tonSendPingReq(
				in := FALSE
			);
		END_IF;

		IF
			stMqttSettings.stMqttSendTelegram.nDataLength > 0
			AND NOT stMqttSettings.bDisconnect
			AND NOT stMqttSettings.bError
			AND stMqttSettings.bSocketConnection
			AND NOT bBusy
		THEN
			iState := C_SEND;
		END_IF;

		IF
			stMqttSettings.bDisconnect
			OR stMqttSettings.bError
			OR NOT stMqttSettings.bSocketConnection
		THEN
			iState := C_STARTUP;
		END_IF;

		(* ensure at least 1 cycle pause *)
		(* bBusy := FALSE; *)

	ELSE
		iState := C_STARTUP;
END_CASE;

(*	END_FUNCTION_BLOCK	*)
END_FUNCTION_BLOCK

(* POU Intern/FB_Mqtt_Receive_V10, ST *)
(* @NESTEDCOMMENTS := 'Yes' *)
(* @PATH := '\/_Generic\/Mqtt\/Intern' *)
(* @OBJECTFLAGS := '0, 8' *)
(* @SYMFILEFLAGS := '2048' *)
FUNCTION_BLOCK FB_Mqtt_Receive_V10
VAR_OUTPUT
	bBusy	: BOOL := FALSE;
END_VAR
VAR_IN_OUT
	stMqttSettings	: ST_MqttSettings;
END_VAR
VAR
	fbSocketReceive		: FB_SocketReceive;
	fbMqttDecodeLength	: FB_Mqtt_DecodeLength_V10;
	stReceiveBuffer		: ST_MqttTelegram;

	iState 			: INT := 0;
	iLengthPosition	: INT := 0;
	index			: INT := 0;
	dwDataLength	: DWORD := 0;
	wTopicLength	: WORD := 0;
	dwValueLength	: DWORD := 0;
END_VAR
VAR CONSTANT
	C_STARTUP				: INT := 0;
	C_RECEIVE_HEADER		: INT := 100;
	C_RECEIVE_HEADER_WAIT	: INT := 110;
	C_RECEIVE_LENGTH		: INT := 120;
	C_RECEIVE_LENGTH_WAIT	: INT := 130;
	C_RECEIVE_DATA			: INT := 200;
	C_RECEIVE_DATA_WAIT		: INT := 210;
	C_IDLE					: INT := 500;
END_VAR

(* @END_DECLARATION := '0' *)
CASE iState OF
	C_STARTUP:
		bBusy 			:= FALSE;
		iLengthPosition	:= 0;
		index			:= 0;
		dwDataLength	:= 0;
		wTopicLength	:= 0;
		dwValueLength	:= 0;
		ClearReceivedPublishTelegram();

		IF
			NOT stMqttSettings.bDisconnect
			AND NOT stMqttSettings.bError
			AND stMqttSettings.bSocketConnection
		THEN
			iState := C_IDLE;
		END_IF;

	(* start receive header *)
	C_RECEIVE_HEADER:
		bBusy := TRUE;
		ClearReceivedPublishTelegram();

		fbSocketReceive(
			bExecute := FALSE
		);

		fbSocketReceive(
			sSrvNetId	:= '',
			hSocket		:= stMqttSettings.hSocket,
			cbLen		:= 2,
			pDest		:= ADR(stReceiveBuffer.arMqttData),
			bExecute 	:= TRUE
		);

		iState := C_RECEIVE_HEADER_WAIT;

	(* wait for header with length *)
	C_RECEIVE_HEADER_WAIT:
		fbSocketReceive(
			bExecute := FALSE
		);

		IF
			NOT fbSocketReceive.bBusy
			AND NOT fbSocketReceive.bError
			AND fbSocketReceive.nRecBytes = 2
		THEN
			iLengthPosition	:= 0;
			stMqttSettings.stMqttReceivedTelegram.arMqttData[0] := stReceiveBuffer.arMqttData[0];
			stMqttSettings.stMqttReceivedTelegram.arMqttData[1] := stReceiveBuffer.arMqttData[1];

			IF stMqttSettings.stMqttReceivedTelegram.arMqttData[1].7 = 1 THEN
				(* payload longer then 127 byte *)
				iLengthPosition := iLengthPosition + 1;
				iState			:= C_RECEIVE_LENGTH;
			ELSE
				IF stMqttSettings.stMqttReceivedTelegram.arMqttData[1] = 0 THEN
					(* no payload received *)
					stMqttSettings.stMqttReceivedTelegram.nDataLength := 2;

					(* copy last telegram *)
					FC_Mqtt_CopyTelegram_V10(
						stMqttSrcTelegram	:= stMqttSettings.stMqttReceivedTelegram,
						stMqttDestTelegram	:= stMqttSettings.stMqttLastReceivedTelegram,
						stMqttSettings		:= stMqttSettings
					);

					iState	:= C_IDLE;
					bBusy 	:= FALSE;
				ELSE
					iState := C_RECEIVE_DATA;
				END_IF;
			END_IF;
		END_IF;

		IF fbSocketReceive.bError THEN
			iState 					:= C_STARTUP;
			stMqttSettings.bError	:= TRUE;
		END_IF;

		IF fbSocketReceive.nRecBytes = 0 THEN
			iState	:= C_IDLE;
			bBusy	:= FALSE;
		END_IF;

		IF
			NOT stMqttSettings.bActive
			OR NOT stMqttSettings.bSocketConnection
		THEN
			iState := C_STARTUP;
		END_IF;

	(* read next remaining length *)
	C_RECEIVE_LENGTH:
		fbSocketReceive(
			bExecute := FALSE
		);

		fbSocketReceive(
			sSrvNetId	:= '',
			hSocket		:= stMqttSettings.hSocket,
			cbLen		:= 1,
			pDest		:= ADR(stReceiveBuffer.arMqttData),
			bExecute 	:= TRUE
		);

		iState := C_RECEIVE_LENGTH_WAIT;

	(* wait for remaining length *)
	C_RECEIVE_LENGTH_WAIT:
		fbSocketReceive(
			bExecute := FALSE
		);

		IF
			NOT fbSocketReceive.bBusy
			AND NOT fbSocketReceive.bError
			AND fbSocketReceive.nRecBytes = 1
		THEN
			stMqttSettings.stMqttReceivedTelegram.arMqttData[1 + iLengthPosition] := stReceiveBuffer.arMqttData[0];

			IF stMqttSettings.stMqttReceivedTelegram.arMqttData[1 + iLengthPosition].7 = 1 THEN
				(* read next length byte *)
				iLengthPosition := iLengthPosition + 1;
				iState			:= C_RECEIVE_LENGTH;

				(* Not more the 4 length bytes *)
				IF iLengthPosition > 4 THEN
					iState 					:= C_STARTUP;
					stMqttSettings.bError	:= TRUE;
				END_IF;
			ELSE
				iState := C_RECEIVE_DATA;
			END_IF;
		END_IF;

		IF fbSocketReceive.bError THEN
			iState 					:= C_STARTUP;
			stMqttSettings.bError	:= TRUE;
		END_IF;

		IF
			NOT stMqttSettings.bActive
			OR NOT stMqttSettings.bSocketConnection
		THEN
			iState := C_STARTUP;
		END_IF;

	(* receive remaining data *)
	C_RECEIVE_DATA:
		fbMqttDecodeLength(
			stMqttTelegram	:= stMqttSettings.stMqttReceivedTelegram,
			dwLength		=> dwDataLength
		);

		fbSocketReceive(
			bExecute := FALSE
		);

		fbSocketReceive(
			sSrvNetId	:= '',
			hSocket		:= stMqttSettings.hSocket,
			cbLen		:= dwDataLength,
			pDest		:= ADR(stReceiveBuffer.arMqttData),
			bExecute 	:= TRUE
		);

		iState := C_RECEIVE_DATA_WAIT;

	(* receive *)
	C_RECEIVE_DATA_WAIT:
		fbSocketReceive(
			bExecute := FALSE
		);

		IF
			NOT fbSocketReceive.bBusy
			AND NOT fbSocketReceive.bError
			AND fbSocketReceive.nRecBytes > 0
		THEN
			MEMCPY(
				destAddr	:= ADR(stMqttSettings.stMqttReceivedTelegram.arMqttData[2 + iLengthPosition]),
			    srcAddr		:= ADR(stReceiveBuffer.arMqttData),
				n  			:= fbSocketReceive.nRecBytes
			);
			stMqttSettings.stMqttReceivedTelegram.nDataLength := 2 + iLengthPosition + fbSocketReceive.nRecBytes;

			(* copy last telegram *)
			FC_Mqtt_CopyTelegram_V10(
				stMqttSrcTelegram	:= stMqttSettings.stMqttReceivedTelegram,
				stMqttDestTelegram	:= stMqttSettings.stMqttLastReceivedTelegram,
				stMqttSettings		:= stMqttSettings
			);

			(* check for publish *)
			IF (stMqttSettings.stMqttReceivedTelegram.arMqttData[0] AND 48) = 48 THEN
				ClearReceivedPublishTelegram();

				(* Length MSB/LSB Topic *)
				wTopicLength :=
						SHL(BYTE_TO_WORD(stMqttSettings.stMqttReceivedTelegram.arMqttData[2 + iLengthPosition + 1]), 8) +
						BYTE_TO_WORD(stMqttSettings.stMqttReceivedTelegram.arMqttData[1 + iLengthPosition + 1]);
				wTopicLength := BE16_TO_HOST(wTopicLength);

				(* Copy topic *)
				MEMCPY(
					destAddr	:= ADR(stMqttSettings.stMqttReceivedPublishTelegram.sTopic),
				    srcAddr		:= ADR(stMqttSettings.stMqttReceivedTelegram.arMqttData[3 + iLengthPosition + 1]),
					n  			:= wTopicLength
				);

				(* Copy value *)
				(* value length = remaining data length - length topic value - 2 byte topic length *)
				dwValueLength := dwDataLength - wTopicLength - 2;

				MEMCPY(
					destAddr	:= ADR(stMqttSettings.stMqttReceivedPublishTelegram.sValue),
				    srcAddr		:= ADR(stMqttSettings.stMqttReceivedTelegram.arMqttData[3 + iLengthPosition + 1 + wTopicLength]),
					n  			:= dwValueLength
				);

				stMqttSettings.stMqttReceivedPublishTelegram.bHasData := TRUE;
			END_IF;

			iState	:= C_IDLE;
			bBusy	:= FALSE;
		END_IF;

		IF fbSocketReceive.bError THEN
			iState 					:= C_STARTUP;
			stMqttSettings.bError	:= TRUE;
		END_IF;

		IF
			NOT stMqttSettings.bActive
			OR NOT stMqttSettings.bSocketConnection
		THEN
			iState := C_STARTUP;
		END_IF;

	(* idle *)
	C_IDLE:
		IF
			NOT stMqttSettings.bDisconnect
			AND NOT stMqttSettings.bError
			AND stMqttSettings.bSocketConnection
			AND NOT bBusy
		THEN
			iState := C_RECEIVE_HEADER;
		END_IF;

		IF
			stMqttSettings.bDisconnect
			OR stMqttSettings.bError
			OR NOT stMqttSettings.bSocketConnection
		THEN
			iState := C_STARTUP;
		END_IF;

		(* ensure at least 1 cycle pause *)
		(* bBusy := FALSE; *)

	ELSE
		iState := C_STARTUP;
END_CASE;

(*	END_FUNCTION_BLOCK	*)
END_FUNCTION_BLOCK
ACTION ClearReceivedPublishTelegram:
MEMSET(
	destAddr	:= ADR(stMqttSettings.stMqttReceivedPublishTelegram.sTopic),
	fillByte  	:= 0,
	n			:= 255
);
stMqttSettings.stMqttReceivedPublishTelegram.sTopic := '';

MEMSET(
	destAddr	:= ADR(stMqttSettings.stMqttReceivedPublishTelegram.sValue),
	fillByte  	:= 0,
	n			:= 255
);
stMqttSettings.stMqttReceivedPublishTelegram.sValue := '';

stMqttSettings.stMqttReceivedPublishTelegram.bHasData := FALSE;
END_ACTION

(* POU Intern/FB_Mqtt_DecodeLength_V10, ST *)
(* @NESTEDCOMMENTS := 'Yes' *)
(* @PATH := '\/_Generic\/Mqtt\/Intern' *)
(* @OBJECTFLAGS := '0, 8' *)
(* @SYMFILEFLAGS := '2048' *)
FUNCTION_BLOCK FB_Mqtt_DecodeLength_V10
VAR_INPUT
	stMqttTelegram : ST_MqttTelegram;
END_VAR
VAR_OUTPUT
	dwLength	: DWORD;
	bAmount		: BYTE;
END_VAR
VAR
	index			: INT;
	diMultiplier	: DINT;
	dwValue			: DWORD;
END_VAR
(* @END_DECLARATION := '0' *)
index			:= 0;
diMultiplier	:= 1;
dwValue			:= 0;

REPEAT
	index := index + 1;

	dwValue := dwValue + (stMqttTelegram.arMqttData[index] AND 127) * diMultiplier;
	diMultiplier := diMultiplier * 128;

	IF diMultiplier > 128*128*128 THEN
		dwLength	:= 0;
		bAmount		:= 0;
		RETURN;
	END_IF;
UNTIL stMqttTelegram.arMqttData[index].7 = 0
END_REPEAT;

dwLength	:= dwValue;
bAmount		:= INT_TO_BYTE(index);

(*
multiplier = 1
value = 0

do
	encodedByte = 'next byte from stream'
	value += (encodedByte AND 127) * multiplier
	multiplier *= 128

	if (multiplier > 128*128*128)
		throw Error(Malformed Remaining Length)
while ((encodedByte AND 128) != 0)

*)

(*	END_FUNCTION_BLOCK	*)
END_FUNCTION_BLOCK

(* POU FB_Mqtt_Publish_V10, ST *)
(* @NESTEDCOMMENTS := 'Yes' *)
(* @PATH := '\/_Generic\/Mqtt' *)
(* @OBJECTFLAGS := '0, 8' *)
(* @SYMFILEFLAGS := '2048' *)
FUNCTION_BLOCK FB_Mqtt_Publish_V10
VAR_INPUT
	sTopic	: STRING[255];
	sValue	: STRING[255];
	bRetain	: BOOL := TRUE;
END_VAR
VAR_OUTPUT
	bBusy	: BOOL := FALSE;
END_VAR
VAR_IN_OUT
	stMqttSettings	: ST_MqttSettings;
END_VAR
VAR
	bFirstPublishDone	: BOOL := FALSE;
	bMustPublish		: BOOL := FALSE;
	sLastValue			: STRING[255];
	iState 				: INT := 0;
	iLengthTopic		: INT := 0;
	iLengthValue		: INT := 0;
	wTopicLength		: WORD;
	stMqttTelegram		: ST_MqttTelegram;
	fbMqttEncodeLength	: FB_Mqtt_EncodeLength_V10;
	bLength1			: BYTE;
	bLength2			: BYTE;
	bLength3			: BYTE;
	bLength4			: BYTE;
	bLengthAmount		: BYTE;
END_VAR
VAR CONSTANT
	C_STARTUP			: INT := 0;
	C_BUILD_TELEGRAM	: INT := 100;
	C_SEND_WAIT			: INT := 110;
	C_IDLE				: INT := 500;
END_VAR
(* @END_DECLARATION := '0' *)
CASE iState OF
	C_STARTUP:
		bFirstPublishDone	:= FALSE;
		bBusy				:= FALSE;

		IF stMqttSettings.bValidConnection THEN
			iState := C_IDLE;
		END_IF;

	(* build publish telegram *)
	C_BUILD_TELEGRAM:
		bBusy := TRUE;
		iLengthTopic := LEN(sTopic);
		iLengthValue := LEN(sValue);

		FC_Mqtt_ClearTelegram_V10(
			stMqttTelegram	:= stMqttTelegram,
			stMqttSettings	:= stMqttSettings
		);

		wTopicLength := iLengthTopic;
		wTopicLength := HOST_TO_BE16(wTopicLength);

		(* Calculate length *)
		(* 2 byte length topic, x byte length topic, x byte length value *)
		fbMqttEncodeLength(
			dwLength := 2 + iLengthTopic + iLengthValue,
			bLength1 => bLength1,
			bLength2 => bLength2,
			bLength3 => bLength3,
			bLength4 => bLength4,
			bAmount	 => bLengthAmount
		);

		(* MQTT Control Packet type, no DUP, no QoS, Retain *)
		stMqttTelegram.arMqttData[0] := 48;
		IF bRetain THEN
			stMqttTelegram.arMqttData[0].0 := 1;
		END_IF;

		(* Remaining Length *)
		CASE bLengthAmount OF
			1:
				stMqttTelegram.arMqttData[1] := bLength1;

			2:
				stMqttTelegram.arMqttData[1] := bLength1;
				stMqttTelegram.arMqttData[2] := bLength2;

			3:
				stMqttTelegram.arMqttData[1] := bLength1;
				stMqttTelegram.arMqttData[2] := bLength2;
				stMqttTelegram.arMqttData[3] := bLength3;

			4:
				stMqttTelegram.arMqttData[1] := bLength1;
				stMqttTelegram.arMqttData[2] := bLength2;
				stMqttTelegram.arMqttData[3] := bLength3;
				stMqttTelegram.arMqttData[4] := bLength4;

			ELSE
				iState 					:= C_STARTUP;
				stMqttSettings.bError	:= TRUE;
		END_CASE;

		(* Length MSB Topic *)
		stMqttTelegram.arMqttData[1 + bLengthAmount] := WORD_TO_BYTE(wTopicLength);
		(* Length LSB Topic *)
		stMqttTelegram.arMqttData[2 + bLengthAmount] := WORD_TO_BYTE(SHR(wTopicLength, 8));

		(* Add topic *)
		MEMCPY(
			destAddr	:= ADR(stMqttTelegram.arMqttData[3 + bLengthAmount]),
		    srcAddr		:= ADR(sTopic),
			n  			:= iLengthTopic
		);

		(* Add Payload *)
		MEMCPY(
			destAddr	:= ADR(stMqttTelegram.arMqttData[3 + bLengthAmount + iLengthTopic]),
		    srcAddr		:= ADR(sValue),
			n  			:= iLengthValue
		);

		(* 1 byte header, x byte variable length, 2 byte topic lenght, x byte topic, x byte value *)
		stMqttTelegram.nDataLength := 1 + bLengthAmount + 2 + iLengthTopic + iLengthValue;

		iState := C_SEND_WAIT;

	(* send telegram *)
	C_SEND_WAIT:
		IF stMqttSettings.stMqttSendTelegram.nDataLength = 0 THEN
			FC_Mqtt_CopyTelegram_V10(
				stMqttSrcTelegram	:= stMqttTelegram,
				stMqttDestTelegram	:= stMqttSettings.stMqttSendTelegram,
				stMqttSettings		:= stMqttSettings
			);

			iState				:= C_IDLE;
			bFirstPublishDone	:= TRUE;
			sLastValue			:= sValue;
		END_IF;

		IF NOT stMqttSettings.bValidConnection THEN
			iState := C_STARTUP;
		END_IF;

	(* idle *)
	C_IDLE:
		bBusy 			:= FALSE;
		bMustPublish 	:= sLastValue <> sValue;

		IF
			stMqttSettings.bValidConnection
			AND (
				bMustPublish
				OR NOT bFirstPublishDone
			)
		THEN
			iState := C_BUILD_TELEGRAM;
		END_IF;

		IF NOT stMqttSettings.bValidConnection THEN
			iState := C_STARTUP;
		END_IF;

	ELSE
		iState := C_STARTUP;
END_CASE;

(*	END_FUNCTION_BLOCK	*)
END_FUNCTION_BLOCK

(* POU Sensors, ST *)
PROGRAM Sensors
VAR
END_VAR
iobroker.Temp_vent_in:=WORD_TO_REAL(HW_temp_vent_in)/10;		(*Temperature pritoka*)

iobroker.Kitchen_room_tempout:=WORD_TO_REAL(HW_temp_street);
IF (iobroker.Kitchen_room_tempout/10>1000)  THEN
	iobroker.Kitchen_room_tempout:=iobroker.Kitchen_room_tempout-65535;
	iobroker.Kitchen_room_tempout:=iobroker.Kitchen_room_tempout/10;
ELSE
	iobroker.Kitchen_room_tempout:=iobroker.Kitchen_room_tempout/10; 	(*Temperature okno*)
END_IF
END_PROGRAM

(* POU RS485read, ST *)
PROGRAM RS485read
VAR
	timeoutvalue					: TIME := T#500ms;		(* timeout while waiting for an answer of the modbus slave *)
	delta_sensor_hum				: INT:=14;					(*Корректировка показаний датчика, % относительной влажности*)
	Period_steam				: INT := 60; 				(* Частота изменения уставки мощности  увлажнителя, секунды*)
	Period_modbus				: INT := 10;  				(* Частота опроса устройств modbus, секунды*)

	r_Target_hum					: REAL;
	r_room_hum					: REAL;
	i_Steam_level				: INT:=0;
	MBdata						: ARRAY [1..2] OF WORD;		(* The size of this array can be adapted to the modbus slaves register area *)




	FtrigBusy					: F_TRIG;
	state						: INT;
	busy						: BOOL;
	LastErrorstate					: INT;
	LastModbusError				: ST_ModbusErrorDiagnostics;
	CounterError					: DINT;
	CounterSuccess				: DINT;
	Timer1						: TON;
	Timer1Q						: BOOL;
	Hum_old						: REAL;
	Steam_response				: WORD:=0;
	Timer2						: TON;
	Timer2Q						: BOOL;
	tTimerValue					: TIME;
	tTimerValue_modbus			: TIME;
	get_run_Merc200_done		: BOOL;
	get_hist_Merc200_done		: BOOL;
	get_run_Merc200				: FB_GET_RUN_MERC200;
	get_hist_Merc200				: FB_GET_HIST_MERC200;

	tmCheck: TON;
END_VAR
tmcheck();
CASE state OF
	0:
		MB.ReadRegs(Execute:= FALSE);
		state := 2;


	2:	(* Kitchen_room Temperature and Humidity *)
		Clear(Buffer := RxBufferCom1);
		MB.ReadRegs(
			UnitID:= 16#01, (* station address *)
			Quantity:= 2,
			MBAddr:= 0,
			cbLength:= 6,
			pMemoryAddr:= ADR(MBdata),
			Execute:= TRUE,
			Timeout:= timeoutvalue,
			Busy => busy,
		);
		IF NOT busy THEN
			IF (mb.Error = FALSE ) THEN
				iobroker.Kitchen_room_temp:=WORD_TO_REAL(MBdata[1])/10;
				iobroker.Kitchen_room_hum:=WORD_TO_REAL(MBdata[2])/10 - delta_sensor_hum;
				MB.ReadRegs(Execute:= FALSE);
				state := 3;
			END_IF
			MB.ReadRegs(Execute:= FALSE);
			state :=3;
		END_IF

	3:	(* Bed_room Temperature and Humidity  *)
		MB.ReadRegs(
			UnitID:= 16#02, (* station address *)
			Quantity:= 2,
			MBAddr:= 0,
			cbLength:= 6,
			pMemoryAddr:= ADR(MBdata),
			Execute:= TRUE,
			Timeout:= timeoutvalue,
			Busy => busy	);
		IF NOT busy THEN
			IF (mb.Error = FALSE ) THEN
				iobroker.Bed_room_temp:=WORD_TO_REAL(MBdata[1])/10;
				iobroker.Bed_room_hum:=WORD_TO_REAL(MBdata[2])/10 - delta_sensor_hum;
				MB.ReadRegs(Execute:= FALSE);
				state := 4;
			END_IF
			MB.ReadRegs(Execute:= FALSE);
			state := 4;
		END_IF

	4:	(* Child_big_room  Temperature and Humidity *)
		MB.ReadRegs(
			UnitID:= 16#03, (* station address *)
			Quantity:= 2,
			MBAddr:= 0,
			cbLength:= 6,
			pMemoryAddr:= ADR(MBdata),
			Execute:= TRUE,
			Timeout:= timeoutvalue,
			Busy => busy	);
		IF NOT busy THEN
			IF (mb.Error = FALSE ) THEN
				iobroker.Child_big_room_temp:=WORD_TO_REAL(MBdata[1])/10;
				iobroker.Child_big_room_hum:=WORD_TO_REAL(MBdata[2])/10 - delta_sensor_hum;
				MB.ReadRegs(Execute:= FALSE);
				state := 5;
			END_IF
			MB.ReadRegs(Execute:= FALSE);
			state := 5;

		END_IF

	5:	(*  Child_small_room Temperature and Humidity *)
		MB.ReadRegs(
			UnitID:= 55, (* station address *)
			Quantity:= 2,
			MBAddr:= 0,
			cbLength:= 6,
			pMemoryAddr:= ADR(MBdata),
			Execute:= TRUE,
			Timeout:= timeoutvalue,
			Busy => busy	);
		IF NOT busy THEN
			IF (mb.Error = FALSE ) THEN
				iobroker.Child_small_room_temp:=WORD_TO_REAL(MBdata[1])/10;
				iobroker.Child_small_room_hum:=WORD_TO_REAL(MBdata[2])/10 - delta_sensor_hum;
				MB.ReadRegs(Execute:= FALSE);
				state := 26;
			END_IF
			MB.ReadRegs(Execute:= FALSE);
			state := 26;

		END_IF

	26:	(* Kitchen_room CO2 *)
		MB.ReadInputRegs(
			UnitID:= 16#68, (* station address *)
			Quantity:= 1,
			MBAddr:= 3,
			cbLength:= 4,
			pMemoryAddr:= ADR(MBdata),
			Execute:= TRUE,
			Timeout:= timeoutvalue,
			Busy => busy	);
		IF NOT busy THEN
			IF (mb.Error = FALSE ) THEN
				iobroker.Kitchen_room_CO2:=WORD_TO_REAL(MBdata[1]);
			END_IF
			MB.ReadRegs(Execute:= FALSE);
			state := 27;
		END_IF

	27:	(* Bed_room CO2  *)
		MB.ReadInputRegs(
			UnitID:= 101, (* station address *)
			Quantity:= 1,
			MBAddr:= 3,
			cbLength:= 4,
			pMemoryAddr:= ADR(MBdata),
			Execute:= TRUE,
			Timeout:= timeoutvalue,
			Busy => busy	);
		IF NOT busy THEN
			IF (mb.Error = FALSE ) THEN
				iobroker.Bed_room_CO2:=WORD_TO_REAL(MBdata[1]);
			END_IF
			MB.ReadRegs(Execute:= FALSE);
			state := 28;
		END_IF

	28:	(* Child_big_room CO2 *)
		MB.ReadInputRegs(
			UnitID:= 102, (* station address *)
			Quantity:= 1,
			MBAddr:= 3,
			cbLength:= 4,
			pMemoryAddr:= ADR(MBdata),
			Execute:= TRUE,
			Timeout:= timeoutvalue,
			Busy => busy	);
		IF NOT busy THEN
			IF (mb.Error = FALSE ) THEN
				iobroker.Child_big_room_CO2:=WORD_TO_REAL(MBdata[1]);
			END_IF
			MB.ReadRegs(Execute:= FALSE);
			state := 29;
		END_IF

	29:	(* Child_small_room CO2  *)
		MB.ReadInputRegs(
			UnitID:= 103, (* station address *)
			Quantity:= 1,
			MBAddr:= 3,
			cbLength:= 4,
			pMemoryAddr:= ADR(MBdata),
			Execute:= TRUE,
			Timeout:= timeoutvalue,
			Busy => busy	);
		IF NOT busy THEN
			IF (mb.Error = FALSE ) THEN
				iobroker.Child_small_room_CO2:=WORD_TO_REAL(MBdata[1]);
			END_IF
			MB.ReadRegs(Execute:= FALSE);
			state := 47;
		END_IF

	47:	(*Изменение уставки мощности увлажнителя при необходимости с частотой Period_steam *)

		IF (iobroker.Steam=TRUE AND iobroker.Vent=TRUE ) THEN
			r_Target_hum:=INT_TO_REAL( iobroker.Target_Hum) ;
			r_room_hum:=iobroker.Bed_room_hum;
			tTimerValue := DINT_TO_TIME(Period_steam*1000);
			Timer2(IN:=NOT Timer2Q , PT:=tTimerValue , Q=>Timer2Q , ET=> );
			IF timer2.q THEN
				IF  ( r_room_hum <= r_Target_hum*0.5 AND i_Steam_level< 50 ) THEN
					i_Steam_level:=50;
				END_IF

				IF ( ( r_room_hum <=   Hum_old )
				AND ( r_room_hum > r_Target_hum*0.5)
				AND ( r_room_hum < r_Target_hum*0.95 )) THEN
					i_Steam_level:=i_Steam_level+1;
				END_IF

				IF ( r_room_hum >= r_Target_hum*1.05) THEN
					i_Steam_level:=i_Steam_level-1;
				END_IF

				Hum_old:=r_room_hum;

			END_IF

			IF (i_Steam_level>100) THEN
				i_Steam_level:=100;
			END_IF

			IF (i_Steam_level<10) THEN
				i_Steam_level:=10;
			END_IF

			iobroker.Steam_level:=INT_TO_BYTE(i_Steam_level);

			MB.WriteSingleRegister(
					UnitID:= 16#0A, (* station address *)
					Quantity:= 1,
					MBAddr:= 1537,
					cbLength:= 2,
					pMemoryAddr:= ADR(iobroker.Steam_level),
					Execute:= TRUE,
					Timeout:= timeoutvalue,
					Busy => busy	);
			IF NOT busy THEN
					MB.WriteSingleRegister(Execute:= FALSE);
					state := 77;
			END_IF
		ELSE
			iobroker.Steam_level:=0;
			state := 77;
		END_IF


	77:		(* Фактический процент текущей  мощности увлажнителя *)

			MB.ReadRegs(
					UnitID:= 16#0A, (* station address *)
					Quantity:= 1,
					MBAddr:= 261,
					cbLength:= 2,
					pMemoryAddr:= ADR(Steam_response),
					Execute:= TRUE,
					Timeout:= timeoutvalue,
					Busy => busy	);
				IF NOT busy THEN
					IF (mb.Error = FALSE ) THEN
						iobroker.Steam_real:=Steam_response;
					END_IF
					MB.ReadRegs(Execute:= FALSE);
					state := 78;

				END_IF


	78:	(* Контрольный датчик Температуры и Влажности*)

			MB.ReadRegs(
			UnitID:= 16#07, (* station address *)
			Quantity:= 2,
			MBAddr:= 0,
			cbLength:= 6,
			pMemoryAddr:= ADR(MBdata),
			Execute:= TRUE,
			Timeout:= timeoutvalue,
			Busy => busy	);
		IF NOT busy THEN
			IF (mb.Error = FALSE ) THEN
				iobroker.Bed_room_temp2:=WORD_TO_REAL(MBdata[1])/10;
				iobroker.Bed_room_hum2:=WORD_TO_REAL(MBdata[2])/10;
				MB.ReadRegs(Execute:= FALSE);
				state := 79;
			END_IF
			MB.ReadRegs(Execute:= FALSE);
			state := 79;

		END_IF
	79:
		tmCheck(in:=FALSE);
		tmCheck(in:=TRUE,pt:=t#2s);
		get_run_Merc200_done := FALSE;
		busy:=TRUE;
		get_run_Merc200( Uv=>iobroker.Uv,Ia=>iobroker.Ia,Pw=>iobroker.Pw, done=>get_run_Merc200_done);
		IF get_run_Merc200_done = TRUE THEN
			busy:=FALSE;
			state:=80;
		ELSIF tmcheck.Q THEN
			busy:=FALSE;
			 state:=80;
		END_IF

	80:
		tmCheck(in:=FALSE);
		tmCheck(in:=TRUE,pt:=t#2s);
		get_hist_Merc200_done := FALSE;
		busy:=TRUE;
		get_hist_Merc200( E_T1=>iobroker.E_T1,E_T2=>iobroker.E_T2,E_T4=>iobroker.E_T4, done=>get_hist_Merc200_done);
		IF get_hist_Merc200_done = TRUE THEN
			busy:=FALSE;
			state:=88;
		ELSIF tmcheck.Q THEN
			busy:=FALSE;
			 state:=88;
		END_IF

	88:
		tTimerValue_modbus := DINT_TO_TIME(Period_modbus*1000);
		Timer1(IN:=NOT Timer1Q , PT:=tTimerValue_modbus , Q=>Timer1Q , ET=> );
		IF timer1.q THEN

		state:=0;
		END_IF

END_CASE

FtrigBusy(CLK:=mb.BUSY );
IF FtrigBusy.Q THEN
	IF mb.Error THEN
		LastModbusError := mb.ErrorDiagnostics;
		LastErrorstate := state;
		CounterError := CounterError + 1;
	ELSE
		CounterSuccess := CounterSuccess + 1;
	END_IF
END_IF

SerialLinecontrolCom1(
	mode:=SerialLinemode_kl6_22b_standard,
	pComIn:=ADR(RS485read.MB.InData),
	pComOut:=ADR(RS485read.MB.OutData),
	SizeComIn:=SIZEOF(RS485read.MB.OutData),
	TxBuffer:=TxBufferCom1,
	RxBuffer:=RxBufferCom1,
	Error=>,
	errorid=>);
END_PROGRAM

(* POU FB_GET_RUN_MERC200, ST *)
FUNCTION_BLOCK FB_GET_RUN_MERC200
VAR_INPUT

END_VAR

VAR_OUTPUT
	Uv				: REAL;
	Ia				: REAL;
	Pw				: REAL;
	done			: BOOL;
END_VAR

VAR
	SendBuffer		: ARRAY[1..7] OF BYTE;
	ReceiveBuffer	: ARRAY[1..14] OF BYTE;
	Clear			: ClearComBuffer;
	state			: INT:= 0;
	tmcheck			: TON;

	crctest			: WORD;
	Uv_word			: WORD;
	Ia_word			: WORD;
	Pw_dword		: DWORD;

	CRC_calc: WORD;
	CRC_get: WORD := 1;

END_VAR
tmcheck();

CASE state OF

0:
	done:=FALSE;
	Clear(Buffer := RxBufferCom1);
	SendBuffer[1] := 16#00;

	SendBuffer[2] := 16#0B; (* Address  dec 740964 = hex 0B 4E 64  *)
	SendBuffer[3] := 16#4E; (* Address *)
	SendBuffer[4] := 16#64; (* Address *)

	SendBuffer[5] := 16#63; (*Command*)
	crctest:=F_CRC16(ADR(SendBuffer), 5);
	MEMCPY(ADR(SendBuffer)+5,ADR(crctest),2);

	SendDataCom1(pSendData:=ADR(SendBuffer),length:=7,TXbuffer:=TXBufferCom1,Busy=>,Error=>);

	tmCheck(in:=FALSE);
	tmCheck(in:=TRUE,pt:=t#2s);
	state:=1;

1: (*ответ*)

	ReceiveDataCom1(pPrefix:=,LenPrefix:=,pSuffix:=,LenSuffix:=,pReceiveData:=ADR(ReceiveBuffer),SizeReceiveData:=14,TImeOut:=t#2s,Reset:=,RXbuffer:=RxBufferCom1,DataReceived=>,busy=>,RxTimeout=>,LenReceiveData=>);

	IF ReceiveDataCom1.Error <> 0 THEN
		state:=9;
	END_IF

	IF ReceiveDataCom1.DataReceived THEN
		state:=2;
	ELSIF tmcheck.Q THEN
		 state:=9;
	END_IF;



2:(*расшифровка*)
	CRC_calc := F_CRC16(ADR(ReceiveBuffer), 12);
	MEMCPY(ADR(CRC_get),ADR(ReceiveBuffer[13]),1);
	MEMCPY(ADR(CRC_get)+1,ADR(ReceiveBuffer[14]),1);


	IF (  ReceiveBuffer[1] = 16#00  AND CRC_calc = CRC_get ) THEN

		MEMCPY(ADR(Uv_word),ADR(ReceiveBuffer[7]),1);
		MEMCPY(ADR(Uv_word)+1,ADR(ReceiveBuffer[6]),1);
(*		Uv:=10*STRING_TO_REAL(BYTE_TO_HEXSTR(ReceiveBuffer[6],1,FALSE))+0.1*STRING_TO_REAL(BYTE_TO_HEXSTR(ReceiveBuffer[7],1,FALSE)); *)
		Uv:=0.1*STRING_TO_REAL(WORD_TO_HEXSTR(Uv_word,1,FALSE));

		MEMCPY(ADR(Ia_word),ADR(ReceiveBuffer[9]),1);
		MEMCPY(ADR(Ia_word)+1,ADR(ReceiveBuffer[8]),1);
(*		Ia:=STRING_TO_REAL(BYTE_TO_HEXSTR(ReceiveBuffer[8],1,FALSE))+0.01*STRING_TO_REAL(BYTE_TO_HEXSTR(ReceiveBuffer[9],1,FALSE)); *)
		Ia:=0.01*STRING_TO_REAL(WORD_TO_HEXSTR(Ia_word,1,FALSE));

		MEMCPY(ADR(Pw_dword),ADR(ReceiveBuffer[12]),1);
		MEMCPY(ADR(Pw_dword)+1,ADR(ReceiveBuffer[11]),1);
		MEMCPY(ADR(Pw_dword)+2,ADR(ReceiveBuffer[10]),1);
		Pw:=STRING_TO_REAL(DWORD_TO_HEXSTR(Pw_dword,1,FALSE));


		state:=10;
	ELSE
		state:=9;
	END_IF

9:
	Uv:=0;
	done := TRUE;
	state:=0;
10:
	done := TRUE;
	state:=0;

END_CASE;
END_FUNCTION_BLOCK

(* POU F_CRC16, ST *)
FUNCTION F_CRC16 : WORD
VAR_INPUT
	pData: POINTER TO BYTE;		(* указатель на блок данных *)
	Size: WORD;						(* размер блока  данных *)
END_VAR
VAR
	Cnt: BYTE;							(* счетчик битов *)
END_VAR
F_CRC16 := 16#FFFF;
WHILE Size > 0 DO
	F_CRC16 := F_CRC16 XOR pData^;
	FOR Cnt := 0 TO 7 DO
		IF F_CRC16.0 = 0 THEN
			F_CRC16 := SHR(F_CRC16, 1);
		ELSE
			F_CRC16 := SHR(F_CRC16, 1) XOR 16#A001;
		END_IF
	END_FOR;
	pData := pData + 1;
	Size := Size - 1;
END_WHILE
END_FUNCTION

(* POU FB_GET_HIST_MERC200, ST *)
FUNCTION_BLOCK FB_GET_HIST_MERC200
VAR_INPUT

END_VAR

VAR_OUTPUT
	E_T1			: REAL;
	E_T2			: REAL;
	E_T3			: REAL;
	E_T4			: REAL;

	done			: BOOL;
END_VAR

VAR
	SendBuffer		: ARRAY[1..7] OF BYTE;
	ReceiveBuffer	: ARRAY[1..23] OF BYTE:=0,0,0,0,0,0,0,0,0,0,0,0,0,0,0,0,0,0,0,0,0,0,0;
	Clear			: ClearComBuffer;
	state			: INT:= 0;
	tmcheck			: TON;

	crctest			: WORD;
	T1_dword		: DWORD;
	T2_dword		: DWORD;
	T3_dword		: DWORD;
	T4_dword		: DWORD;

	CRC_calc: WORD;
	CRC_get: WORD := 1;

END_VAR
tmcheck();

CASE state OF

0:
	done:=FALSE;
	Clear(Buffer := RxBufferCom1);
	SendBuffer[1] := 16#00;

	SendBuffer[2] := 16#0B; (* Address  dec 740964 =0B 4E 64    *)
	SendBuffer[3] := 16#4E; (* Address *)
	SendBuffer[4] := 16#64; (* Address *)

	SendBuffer[5] := 16#27; (*Command*)

	crctest:=F_CRC16(ADR(SendBuffer), 5);
	MEMCPY(ADR(SendBuffer)+5,ADR(crctest),2);

	SendDataCom1(pSendData:=ADR(SendBuffer),length:=7,TXbuffer:=TXBufferCom1,Busy=>,Error=>);

	tmCheck(in:=FALSE);
	tmCheck(in:=TRUE,pt:=t#2s);
	state:=1;

1: (*ответ*)

	ReceiveDataCom1(pPrefix:=,LenPrefix:=,pSuffix:=,LenSuffix:=,pReceiveData:=ADR(ReceiveBuffer),SizeReceiveData:=23,TImeOut:=t#2s,Reset:=,RXbuffer:=RxBufferCom1,DataReceived=>,busy=>,RxTimeout=>,LenReceiveData=>);

	IF ReceiveDataCom1.Error <> 0 THEN
		state:=9;
	END_IF

	IF ReceiveDataCom1.DataReceived THEN
		state:=2;
	ELSIF tmcheck.Q THEN
		 state:=9;
	END_IF;



2:(*расшифровка*)
	CRC_calc := F_CRC16(ADR(ReceiveBuffer), 21);
	MEMCPY(ADR(CRC_get),ADR(ReceiveBuffer[22]),1);
	MEMCPY(ADR(CRC_get)+1,ADR(ReceiveBuffer[23]),1);


	IF (  ReceiveBuffer[1] = 16#00  AND ReceiveBuffer[2] = 16#0B AND ReceiveBuffer[3] = 16#4E AND ReceiveBuffer[4] = 16#64  AND ReceiveBuffer[5] = 16#27) THEN

		MEMCPY(ADR(T1_dword),ADR(ReceiveBuffer[9]),1);
		MEMCPY(ADR(T1_dword)+1,ADR(ReceiveBuffer[8]),1);
		MEMCPY(ADR(T1_dword)+2,ADR(ReceiveBuffer[7]),1);
		MEMCPY(ADR(T1_dword)+3,ADR(ReceiveBuffer[6]),1);
		E_T1:=0.01*STRING_TO_REAL(DWORD_TO_HEXSTR(T1_dword,1,FALSE));

		MEMCPY(ADR(T2_dword),ADR(ReceiveBuffer[13]),1);
		MEMCPY(ADR(T2_dword)+1,ADR(ReceiveBuffer[12]),1);
		MEMCPY(ADR(T2_dword)+2,ADR(ReceiveBuffer[11]),1);
		MEMCPY(ADR(T2_dword)+3,ADR(ReceiveBuffer[10]),1);
		E_T2:=0.01*STRING_TO_REAL(DWORD_TO_HEXSTR(T2_dword,1,FALSE));

		MEMCPY(ADR(T3_dword),ADR(ReceiveBuffer[17]),1);
		MEMCPY(ADR(T3_dword)+1,ADR(ReceiveBuffer[16]),1);
		MEMCPY(ADR(T3_dword)+2,ADR(ReceiveBuffer[15]),1);
		MEMCPY(ADR(T3_dword)+3,ADR(ReceiveBuffer[14]),1);
		E_T3:=0.01*STRING_TO_REAL(DWORD_TO_HEXSTR(T3_dword,1,FALSE));

		MEMCPY(ADR(T4_dword),ADR(ReceiveBuffer[21]),1);
		MEMCPY(ADR(T4_dword)+1,ADR(ReceiveBuffer[20]),1);
		MEMCPY(ADR(T4_dword)+2,ADR(ReceiveBuffer[19]),1);
		MEMCPY(ADR(T4_dword)+3,ADR(ReceiveBuffer[18]),1);
		E_T4:=0.01*STRING_TO_REAL(DWORD_TO_HEXSTR(T4_dword,1,FALSE));

		state:=10;
	ELSE
		state:=9;
	END_IF

9:
	E_T1:=0;
	E_T2:=0;

	done := TRUE;
	state:=0;
10:
	done := TRUE;
	state:=0;

END_CASE;
END_FUNCTION_BLOCK

(* POU VentControl, ST *)
PROGRAM VentControl
VAR
	Temperature_max_to_heat		: REAL:=17;		(* Максимальная температура наружнего воздуха при которой разрешено включать воздухонагреватель *)
	Temperature_min_for_steam	: REAL:=17;		(* Минимальная температура воздуха в вент канале для разрешения работы увлажнителя *)
	gisterezis					: REAL:=0.2;		(* Гистерезис  разрешения включения воздухонагревателя, градусы цельсия *)


END_VAR
(* Состояние приточного клапана *)

IF (HW_sensor_vent_valve_opened=TRUE) THEN
	iobroker.Vent_valve_status:=1;
END_IF

IF (HW_sensor_vent_valve_closed=TRUE) THEN
	iobroker.Vent_valve_status:=0;
END_IF

IF (HW_sensor_vent_valve_closed=FALSE AND HW_sensor_vent_valve_opened=FALSE) THEN
	iobroker.Vent_valve_status:=2;
END_IF


IF (HW_kitchen_button_vent_out=TRUE) THEN	(* Если активирована кнопка надплитной вытяжки*)
	HW_vent_out:=TRUE;						(* Включаем вытяжной вент *)
	HW_vent_out_level:=32767;					(* Подаём управляющий сигнал DC на максимум *)
	HW_kitchen_vent_out:=TRUE;				(* Включаем вент надплитной вытяжки *)
ELSE
	HW_kitchen_vent_out:=FALSE;				(* Оключаем вент надплитной вытяжки *)
	IF (iobroker.Vent_out=FALSE) THEN			(* Если уставка работы вытяжного вента = FALSE*)
		HW_vent_out:=FALSE;					(* Отключаем вытяжной вент *)
	ELSE
		HW_vent_out:=TRUE;					(*  Включаем вытяжной вент  *)
	END_IF
END_IF


IF (iobroker.Vent=FALSE) THEN
	HW_steam:=FALSE;
	HW_vent_in_heat:=FALSE;
	HW_vent_valve:=FALSE;	(* COMMENT THIS LINE TEMPORARY  ЛЕТНИЙ РЕЖИМ  !!!!!!!!!!!!!!!!!!!!!!!!!!!!!!!!!!!*)
	HW_trans_power:=FALSE;
ELSE
	HW_vent_valve:=TRUE;
	IF (HW_sensor_vent_valve_opened=TRUE) THEN
		HW_trans_power:=TRUE;
		IF (HW_vent_reay_pressure=TRUE) THEN
			IF (iobroker.Temp_vent_in>Temperature_min_for_steam) THEN
				HW_steam:=iobroker.Steam;
			ELSE
				HW_steam:=FALSE;
			END_IF
			IF (iobroker.Vent_heat=2) THEN
				IF (iobroker.Kitchen_room_tempout < Temperature_max_to_heat-gisterezis) THEN
					HW_vent_in_heat:=TRUE;
					IF (iobroker.Vent_heat_level=TRUE) THEN
						HW_vent_in_heat_level:=TRUE;
					END_IF
				END_IF
				IF (iobroker.Kitchen_room_tempout > Temperature_max_to_heat+gisterezis) THEN
					HW_vent_in_heat:=FALSE;
				END_IF
			ELSE
				IF (iobroker.Vent_heat=1) THEN
					HW_vent_in_heat:=TRUE;
					IF (iobroker.Vent_heat_level=TRUE) THEN
						HW_vent_in_heat_level:=TRUE;
					ELSE
						HW_vent_in_heat_level:=FALSE;
					END_IF
				END_IF
				IF (iobroker.Vent_heat=0) THEN
					HW_vent_in_heat:=FALSE;
				END_IF
			END_IF
		END_IF (*vent_relay_pressure*)
	END_IF (*vent_valve_opened*)
END_IF (*Vent*)
END_PROGRAM

(* POU VentPower, ST *)
PROGRAM VentPower
VAR
	Vent_power			: REAL:=30;	(* После перезагрузки ПЛК задаём начальную мощность приточного вента - условных 30%  *)
	Vent_power_out		: INT:=30;		(* После перезагрузки ПЛК задаём начальную мощность вытяжного вента - условных 30%  *)
	CO2_old				: REAL:=410;	(* После перезагрузки ПЛК задаём принудительно последнее значение CO2 = 410 (абсолютно свежий воздух) *)
	Period_vent_switch	: INT:=60; (* Период переключения режимов работы вентилятора по показаниям датчиков CO2, секунды*)
	Timer1				: TON;
	Timer1Q				: BOOL;
	count				: INT:=0;
	CO2_max			: REAL;
	tTimerValue			: TIME;



END_VAR
tTimerValue := DINT_TO_TIME(Period_vent_switch*1000);

IF (iobroker.Vent =TRUE OR iobroker.Vent_out=TRUE ) THEN

	Timer1(IN:=NOT Timer1Q , PT:=tTimerValue , Q=>Timer1Q , ET=> );
	IF timer1.q THEN
		CO2_max:=MAX(iobroker.Kitchen_room_CO2, MAX (iobroker.Bed_room_CO2, MAX (iobroker.Child_big_room_CO2, iobroker.Child_small_room_CO2)));
		IF (  (CO2_max >=  CO2_old-10 )  AND ( CO2_max >  INT_TO_REAL(iobroker.Target_CO2)*1.05 ) ) THEN
			Vent_power:=Vent_power+2;
		END_IF
		count:=count+1;
		IF (count = 5)	THEN
			IF (  CO2_max <=  INT_TO_REAL(iobroker.Target_CO2)*0.99) THEN
				Vent_power:=Vent_power-2;
			END_IF
			count:=1;
		END_IF

		IF (Vent_power>80) THEN
			Vent_power:=80;
		END_IF
		IF(Vent_power<20) THEN
			Vent_power:=20;
		END_IF

		IF (Vent_Power > 75  ) THEN
			iobroker.Vent_input_level:=200;									(* 200 м. куб в час при подаче напряжения на приточный вентилятор  220V *)
			HW_vent_in_trans_160_220:=FALSE;
			HW_vent_in_trans_LO_HI:=FALSE;
			IF (HW_kitchen_button_vent_out=FALSE) THEN					(* Если НЕ  работает кухонная надплитная вытяжка, то нужна тонкая регулировка вытяжного вента *)
				HW_vent_out_level:=REAL_TO_WORD(32767*60/100);			(* 200  м. куб в час при подаче x  DC напряжения на вытяжной вентилятор  *)
				Vent_power_out:=45;
			END_IF

			ELSIF (Vent_Power>50 ) THEN

				iobroker.Vent_input_level:=180; 								(* 180/200 м. куб в час при подаче напряжения на приточный вентилятор  220V *)
				HW_vent_in_trans_160_220:=FALSE;
				HW_vent_in_trans_LO_HI:=FALSE;
				IF (HW_kitchen_button_vent_out=FALSE) THEN				(* Если НЕ  работает кухонная надплитная вытяжка, то нужна тонкая регулировка вытяжного вента *)
					HW_vent_out_level:=REAL_TO_WORD(32767*45/100); 		(* 180  м. куб в час при подаче x  DC напряжения на вытяжной вентилятор  *)
					Vent_power_out:=40;
				END_IF


			ELSIF (Vent_Power>35 AND Vent_Power<=50) THEN

					iobroker.Vent_input_level:=150;							 (* 150 м. куб в час при подаче напряжения на приточный вентилятор  160V *)
					HW_vent_in_trans_160_220:=TRUE;
					HW_vent_in_trans_LO_HI:=FALSE;
					IF (HW_kitchen_button_vent_out=FALSE) THEN			(* Если НЕ  работает кухонная надплитная вытяжка, то нужна тонкая регулировка вытяжного вента *)
						HW_vent_out_level:=REAL_TO_WORD(32767*35/100);	(* 150  м. куб в час при подаче x  DC напряжения на вытяжной вентилятор  *)
						Vent_power_out:=35;
					END_IF

			ELSIF (Vent_Power>25 AND Vent_Power<=35) THEN

					iobroker.Vent_input_level:=110; (* 130V*)					 (* 110 м. куб в час при подаче напряжения на приточный вентилятор  130V *)
					HW_vent_in_trans_105_130:=FALSE;
					HW_vent_in_trans_LO_HI:=TRUE;
					IF (HW_kitchen_button_vent_out=FALSE) THEN			(* Если НЕ  работает кухонная надплитная вытяжка, то нужна тонкая регулировка вытяжного вента *)
						HW_vent_out_level:=REAL_TO_WORD(32767*25/100);	(* 110  м. куб в час при подаче x  DC напряжения на вытяжной вентилятор  *)
						Vent_power_out:=25;
					END_IF

			ELSE	(* Vent_Power > 80 *)

				iobroker.Vent_input_level:=80; (* 105V*)						 (* 80 м. куб в час при подаче напряжения на приточный вентилятор  105V *)
				HW_vent_in_trans_105_130:=TRUE;
				HW_vent_in_trans_LO_HI:=TRUE;
				IF (HW_kitchen_button_vent_out=FALSE) THEN				(* Если НЕ  работает кухонная надплитная вытяжка, то нужна тонкая регулировка вытяжного вента *)
					HW_vent_out_level:=REAL_TO_WORD(32767*20/100);		(* 80  м. куб в час при подаче x  DC напряжения на вытяжной вентилятор  *)
					Vent_power_out:=20;
				END_IF


			END_IF	(* Vent_Power > 80 *)
			CO2_old:=CO2_max;
			iobroker.Vent_output_level:=Vent_power_out;
	END_IF	(* Timer1 *)

ELSE	 (* Vent=TRUE*)

	iobroker.Vent_input_level:=0;
	IF (HW_kitchen_button_vent_out=FALSE) THEN
		HW_vent_out_level:=REAL_TO_WORD(32767*20/100);
	END_IF
	iobroker.Vent_output_level:=Vent_power_out;

END_IF   (* Vent=TRUE*)
END_PROGRAM

(* POU Counters, ST *)
PROGRAM Counters
VAR

	Trigger_bathroom_water_warm: F_TRIG;
	Trigger_bathroom_water_cold: F_TRIG;
	Trigger_kitchen_water_warm: F_TRIG;
	Trigger_kitchen_water_cold: F_TRIG;

END_VAR
Trigger_bathroom_water_warm(CLK :=HW_impulse_bathroom_water_warm);
Trigger_bathroom_water_cold(CLK :=HW_impulse_bathroom_water_cold);
Trigger_kitchen_water_warm(CLK :=HW_impulse_kitchen_water_warm);
Trigger_kitchen_water_cold(CLK :=HW_impulse_kitchen_water_cold);

IF (Trigger_bathroom_water_warm.Q) THEN
	iobroker.Bathroom_stat_warm_water:=iobroker.Bathroom_stat_warm_water+1;
	Bathroom_stat_warm_water_mem:=iobroker.Bathroom_stat_warm_water;
END_IF

IF (Trigger_bathroom_water_cold.Q) THEN
	iobroker.Bathroom_stat_cold_water:=iobroker.Bathroom_stat_cold_water+1;
	Bathroom_stat_cold_water_mem:=iobroker.Bathroom_stat_cold_water;
END_IF

IF (Trigger_kitchen_water_warm.Q) THEN
	iobroker.Kitchen_stat_warm_water:=iobroker.Kitchen_stat_warm_water+1;
	Kitchen_stat_warm_water_mem:=iobroker.Kitchen_stat_warm_water;
END_IF

IF (Trigger_kitchen_water_cold.Q) THEN
	iobroker.Kitchen_stat_cold_water:=iobroker.Kitchen_stat_cold_water+1;
	Kitchen_stat_cold_water_mem:=iobroker.Kitchen_stat_cold_water;
END_IF
END_PROGRAM

(* POU Fluid_bath, ST *)
PROGRAM Fluid_bath
VAR
	BUTTON3 	:	 R_TRIG;  (* Конпка №3 - переключение подачи воды в санузлах *)
END_VAR
iobroker.FLD_BATH:=HW_sensor_fld_van;
iobroker.FLD_PRC:=HW_sensor_fld_post;
iobroker.FLD_TLT:=HW_sensor_fld_tlt;


IF (iobroker.FLD_BATH=TRUE OR iobroker.FLD_PRC=TRUE OR iobroker.FLD_TLT=TRUE ) THEN
	HW_valve_water_bathroom:=FALSE;
	iobroker.FLD_valve_bathroom:=FALSE;
	iobroker.FLD_ALRM_BATH:=TRUE;
ELSE
	IF (iobroker.FLD_ALRM_BATH=FALSE) THEN
		HW_valve_water_bathroom:=TRUE;
		iobroker.FLD_valve_bathroom:=TRUE;
	ELSE
		HW_valve_water_bathroom:=FALSE;
		iobroker.FLD_valve_bathroom:=FALSE;
	END_IF
END_IF

BUTTON3 (CLK:=HW_IN03);

IF (     BUTTON3.Q ) THEN
	IF (iobroker.FLD_valve_bathroom=FALSE) THEN
		IF (iobroker.FLD_BATH=FALSE AND iobroker.FLD_PRC=FALSE AND iobroker.FLD_TLT=FALSE) THEN
			HW_valve_water_bathroom:=TRUE;
			iobroker.FLD_valve_bathroom:=TRUE;
			iobroker.FLD_ALRM_BATH:=FALSE;
		END_IF
	ELSE
		iobroker.FLD_ALRM_BATH:=TRUE;
		HW_valve_water_bathroom:=FALSE;
		iobroker.FLD_valve_bathroom:=FALSE;
	END_IF
END_IF
END_PROGRAM

(* POU Fluid_kitchen, ST *)
PROGRAM Fluid_kitchen
VAR
	BUTTON2 	:	 R_TRIG;  (* Конпка №2 - переключение подачи воды в кухне  *)
END_VAR
iobroker.FLD_KUH:=HW_sensor_fld_kitchen;



IF (iobroker.FLD_KUH=TRUE) THEN
	HW_valve_water_kitchen:=FALSE;
	iobroker.FLD_valve_kitchen:=FALSE;
	iobroker.FLD_ALRM_KITCHEN:=TRUE;
ELSE
	IF (iobroker.FLD_ALRM_KITCHEN=FALSE) THEN
		HW_valve_water_kitchen:=TRUE;
		iobroker.FLD_valve_kitchen:=TRUE;
	ELSE
		HW_valve_water_kitchen:=FALSE;
		iobroker.FLD_valve_kitchen:=FALSE;
	END_IF
END_IF

BUTTON2 (CLK:=HW_IN02);

IF ( BUTTON2.Q ) THEN
	IF (HW_valve_water_kitchen=FALSE) THEN
		IF (iobroker.FLD_KUH=FALSE) THEN
			HW_valve_water_kitchen:=TRUE;
			iobroker.FLD_valve_kitchen:=TRUE;
			iobroker.FLD_ALRM_KITCHEN:=FALSE;
		END_IF
	ELSE
		iobroker.FLD_ALRM_KITCHEN:=TRUE;
		HW_valve_water_kitchen:=FALSE;
		iobroker.FLD_valve_kitchen:=FALSE;
	END_IF
END_IF
END_PROGRAM

(* POU Light_hall, ST *)
PROGRAM Light_hall
VAR
	Timer1			: TOF;
	tTimerValue		: TIME;
	Period_light		: INT := 60;		(* Время работы светильника по датчику движения, секунды *)
END_VAR
tTimerValue := DINT_TO_TIME(Period_light*1000);
Timer1(IN:=(NOT HW_PIR_HALL OR NOT HW_PIR_door), PT:=tTimerValue);
(* HW_LIGHT_HALL:=Timer1.Q; *)
END_PROGRAM

(* POU Door, ST *)
PROGRAM Door
VAR
	Timer1			: TOF;
	tTimerValue		: TIME;
	Period_light		: INT := 60;		(* Время работы светильника по датчику движения, секунды *)
END_VAR
tTimerValue := DINT_TO_TIME(Period_light*1000);

IF HW_PIR_HALL THEN
	Timer1(IN:=(NOT HW_gerkon ), PT:=tTimerValue);
	IF  (NOT Timer1.Q AND HW_gerkon) THEN
		(* OUT *)
	END_IF
END_IF
END_PROGRAM

(* POU Fluid, ST *)
PROGRAM Fluid
VAR
END_VAR
iobroker.FLD_BATH:=HW_sensor_fld_van;
iobroker.FLD_KUH:=HW_sensor_fld_kitchen;
iobroker.FLD_PRC:=HW_sensor_fld_post;
iobroker.FLD_TLT:=HW_sensor_fld_tlt;


IF (iobroker.FLD_BATH=TRUE OR iobroker.FLD_PRC=TRUE OR iobroker.FLD_TLT=TRUE ) THEN
	iobroker.FLD_ALRM_BATH:=TRUE;
	HW_valve_water_bathroom:=FALSE;
	iobroker.FLD_valve_bathroom:=FALSE;
END_IF

(*IF (FLD_BATH=FALSE AND FLD_PRC=FALSE AND FLD_TLT=FALSE  AND FLD_ALRM_BATH=FALSE AND FLD_valve_bathroom=TRUE) THEN
	HW_valve_water_bathroom:=TRUE;
END_IF*)

IF (iobroker.FLD_BATH=TRUE OR iobroker.FLD_PRC=TRUE OR  iobroker.FLD_TLT=TRUE  OR  iobroker.FLD_ALRM_BATH=TRUE ) THEN
	iobroker.FLD_valve_bathroom:=FALSE;
END_IF

HW_valve_water_bathroom:=iobroker.FLD_valve_bathroom;

IF (iobroker.FLD_KUH=TRUE ) THEN
	iobroker.FLD_ALRM_KITCHEN:=TRUE;
	HW_valve_water_kitchen:=FALSE;
	iobroker.FLD_valve_kitchen:=FALSE;
END_IF


IF (iobroker.FLD_KUH=TRUE  OR iobroker.FLD_ALRM_KITCHEN=TRUE ) THEN
	iobroker.FLD_valve_kitchen:=FALSE;
END_IF
HW_valve_water_kitchen:=iobroker.FLD_valve_kitchen;
END_PROGRAM

(* POU FB_Mqtt_Subscribe_V10, ST *)
(* @NESTEDCOMMENTS := 'Yes' *)
(* @PATH := '\/_Generic\/Mqtt' *)
(* @OBJECTFLAGS := '0, 8' *)
(* @SYMFILEFLAGS := '2048' *)
FUNCTION_BLOCK FB_Mqtt_Subscribe_V10
VAR_INPUT
	sTopic	: STRING[255];
	bAccept	: BOOL := FALSE; (* When false, subscribe but do not set bNewValue output *)
END_VAR
VAR_OUTPUT
	sValue		: STRING[255];
	bNewValue	: BOOL := FALSE;
	bBusy		: BOOL := FALSE;
END_VAR
VAR_IN_OUT
	stMqttSettings	: ST_MqttSettings;
END_VAR
VAR
	iState 				: INT := 0;
	bSubscribeSent		: BOOL := FALSE;
	bSubAckReceived		: BOOL := FALSE;
	iTopicLength		: INT := 0;
	wTopicLength		: WORD;
	stMqttTelegram		: ST_MqttTelegram;
	fbMqttEncodeLength	: FB_Mqtt_EncodeLength_V10;
	bLength1			: BYTE;
	bLength2			: BYTE;
	bLength3			: BYTE;
	bLength4			: BYTE;
	bLengthAmount		: BYTE;

	wPackageIdentifier			: WORD;
	wTelegramPackageIdentifier	: WORD;
END_VAR
VAR CONSTANT
	C_STARTUP			: INT := 0;
	C_BUILD_TELEGRAM	: INT := 100;
	C_SEND_WAIT			: INT := 110;
	C_CHECK_TELEGRAM	: INT := 200;
	C_IDLE				: INT := 500;
END_VAR

(* @END_DECLARATION := '0' *)
CASE iState OF
	C_STARTUP:
		wPackageIdentifier 	:= 0;
		bSubscribeSent		:= FALSE;
		bSubAckReceived		:= FALSE;
		bNewValue			:= FALSE;
		sValue 				:= '';
		bBusy				:= FALSE;

		IF stMqttSettings.bValidConnection THEN
			iState := C_IDLE;
		END_IF;

	(* build publish telegram *)
	C_BUILD_TELEGRAM:
		bBusy 								:= TRUE;
		wPackageIdentifier 					:= stMqttSettings.wPackageIdentifier;
		stMqttSettings.wPackageIdentifier 	:= stMqttSettings.wPackageIdentifier + 1;
		iTopicLength						:= LEN(sTopic);

		FC_Mqtt_ClearTelegram_V10(
			stMqttTelegram	:= stMqttTelegram,
			stMqttSettings	:= stMqttSettings
		);

		wTopicLength := iTopicLength;
		wTopicLength := HOST_TO_BE16(wTopicLength);

		wTelegramPackageIdentifier := HOST_TO_BE16(wPackageIdentifier);

		(* Calculate length *)
		(* 2 byte package identifier, 2 byte length topic, x byte length topic, 1 byte QoS *)
		fbMqttEncodeLength(
			dwLength := 2 + 2 + iTopicLength + 1,
			bLength1 => bLength1,
			bLength2 => bLength2,
			bLength3 => bLength3,
			bLength4 => bLength4,
			bAmount	 => bLengthAmount
		);

		(* MQTT Control Packet type *)
		stMqttTelegram.arMqttData[0] := 130;

		(* Remaining Length *)
		CASE bLengthAmount OF
			1:
				stMqttTelegram.arMqttData[1] := bLength1;

			2:
				stMqttTelegram.arMqttData[1] := bLength1;
				stMqttTelegram.arMqttData[2] := bLength2;

			3:
				stMqttTelegram.arMqttData[1] := bLength1;
				stMqttTelegram.arMqttData[2] := bLength2;
				stMqttTelegram.arMqttData[3] := bLength3;

			4:
				stMqttTelegram.arMqttData[1] := bLength1;
				stMqttTelegram.arMqttData[2] := bLength2;
				stMqttTelegram.arMqttData[3] := bLength3;
				stMqttTelegram.arMqttData[4] := bLength4;

			ELSE
				iState 					:= C_STARTUP;
				stMqttSettings.bError	:= TRUE;
		END_CASE;

		(* Packet Identifier MSB *)
		stMqttTelegram.arMqttData[1 + bLengthAmount] := WORD_TO_BYTE(wTelegramPackageIdentifier);
		(* Packet Identifier LSB *)
		stMqttTelegram.arMqttData[2 + bLengthAmount] := WORD_TO_BYTE(SHR(wTelegramPackageIdentifier, 8));
		(* Length MSB Topic *)
		stMqttTelegram.arMqttData[3 + bLengthAmount] := WORD_TO_BYTE(wTopicLength);
		(* Length MSB Topic *)
		stMqttTelegram.arMqttData[4 + bLengthAmount] := WORD_TO_BYTE(SHR(wTopicLength, 8));

		(* Add topic *)
		MEMCPY(
			destAddr	:= ADR(stMqttTelegram.arMqttData[5 + bLengthAmount]),
		    srcAddr		:= ADR(sTopic),
			n  			:= iTopicLength
		);

		(* 1 byte header, x byte variable length, 2 byte package identifier, 2 byte topic lenght, x byte topic, 1 byte QoS *)
		stMqttTelegram.nDataLength := 1 + bLengthAmount + 2 + 2 + iTopicLength + 1;

		iState := C_SEND_WAIT;

	(* send telegram *)
	C_SEND_WAIT:
		IF stMqttSettings.stMqttSendTelegram.nDataLength = 0 THEN
			FC_Mqtt_CopyTelegram_V10(
				stMqttSrcTelegram	:= stMqttTelegram,
				stMqttDestTelegram	:= stMqttSettings.stMqttSendTelegram,
				stMqttSettings		:= stMqttSettings
			);

			bSubscribeSent	:= TRUE;
			iState			:= C_IDLE;
		END_IF;

		IF NOT stMqttSettings.bValidConnection THEN
			iState := C_STARTUP;
		END_IF;

	(* check telegram *)
	C_CHECK_TELEGRAM:
		bBusy 			:= TRUE;

		IF
			stMqttSettings.stMqttReceivedPublishTelegram.bHasData
			AND stMqttSettings.stMqttReceivedPublishTelegram.sTopic = sTopic
		THEN
			FC_Mqtt_ClearTelegram_V10(
				stMqttTelegram	:= stMqttSettings.stMqttReceivedTelegram,
				stMqttSettings	:= stMqttSettings
			);
			stMqttSettings.stMqttReceivedPublishTelegram.bHasData := FALSE;

			sValue		:= stMqttSettings.stMqttReceivedPublishTelegram.sValue;
			bNewValue 	:= TRUE;
		END_IF;

		iState := C_IDLE;

	(* idle *)
	C_IDLE:
		bBusy 		:= FALSE;
		bNewValue	:= FALSE;

		IF
			stMqttSettings.bValidConnection
			AND NOT bSubscribeSent
			AND NOT bSubAckReceived
		THEN
			iState := C_BUILD_TELEGRAM;
		END_IF;

		(* Check for correct SubAck *)
		IF
			bSubscribeSent
			AND stMqttSettings.stMqttReceivedTelegram.nDataLength = 5
			AND stMqttSettings.stMqttReceivedTelegram.arMqttData[0] = 144
			AND stMqttSettings.stMqttReceivedTelegram.arMqttData[1] = 3
			AND stMqttSettings.stMqttReceivedTelegram.arMqttData[2] = WORD_TO_BYTE(wTelegramPackageIdentifier)
			AND stMqttSettings.stMqttReceivedTelegram.arMqttData[3] = WORD_TO_BYTE(SHR(wTelegramPackageIdentifier, 8))
			AND stMqttSettings.stMqttReceivedTelegram.arMqttData[4] = 0
		THEN
			FC_Mqtt_ClearTelegram_V10(
				stMqttTelegram	:= stMqttSettings.stMqttReceivedTelegram,
				stMqttSettings	:= stMqttSettings
			);
			bSubAckReceived := TRUE;
		END_IF;

		(* Check for error SubAck *)
		IF
			bSubscribeSent
			AND stMqttSettings.stMqttReceivedTelegram.nDataLength = 5
			AND stMqttSettings.stMqttReceivedTelegram.arMqttData[0] = 144
			AND stMqttSettings.stMqttReceivedTelegram.arMqttData[1] = 3
			AND stMqttSettings.stMqttReceivedTelegram.arMqttData[2] = WORD_TO_BYTE(wTelegramPackageIdentifier)
			AND stMqttSettings.stMqttReceivedTelegram.arMqttData[3] = WORD_TO_BYTE(SHR(wTelegramPackageIdentifier, 8))
			AND stMqttSettings.stMqttReceivedTelegram.arMqttData[4].7 = 1
		THEN
			stMqttSettings.bError := TRUE;
		END_IF;

		(* Check for publish *)
		IF
			bSubAckReceived
			AND stMqttSettings.stMqttReceivedPublishTelegram.bHasData
			AND bAccept
		THEN
			iState := C_CHECK_TELEGRAM;
		END_IF;

		IF NOT stMqttSettings.bValidConnection THEN
			iState := C_STARTUP;
		END_IF;

	ELSE
		iState := C_STARTUP;
END_CASE

(*	END_FUNCTION_BLOCK	*)
END_FUNCTION_BLOCK
